REGION Network 49: Step[1021] : Uw Semi Splicer Vacuum Left Bottom HomePos & Right Bottom WorkPos Command
   RUNG wire#powerrail
      { S7_Templates := "SrcType := DInt" } EQ_Contact(in1 := "Unit1.Em2.ControlNodes".SemiAutuSplice.sequence.status.currentStep, in2 := #JOB_10_STEP_21)
      Contact( "Unit1.Em2.ControlNodes".SemiAutuSplice.sequence.status.seqActive )
      wire#w1
      I_Contact( "Unit1.Em2.ControlNodes".cmUwSemiSplicerVacuumRightBottomOnOff.monitoring.inWorkPos )
      Coil( "Unit1.Em2.ControlNodes".SemiAutuSplice."step".action[1021] )
   END_RUNG
   RUNG wire#w1
      Contact( "Unit1.Em2.ControlNodes".cmUwSemiSplicerVacuumRightBottomOnOff.monitoring.inWorkPos )
      wire#w2
      Contact( "Unit1.Em2.ControlNodes".cmUwSemiSplicerVacuumLeftBottomOnOff.monitoring.inWorkPos )
      wire#w3
      Coil( "Unit1.Em2.ControlNodes".SemiAutuSplice."step".action[1022] )
   END_RUNG
   RUNG wire#w1
      Contact( "Unit1.Em2.HmiInterface".cmUwSemiSplicerVacuumRightBottomOnOff.monitoring.goToWorkPos )
   END_RUNG wire#w2
   RUNG wire#w2
      Contact( "Unit1.Em2.HmiInterface".cmUwSemiSplicerVacuumLeftBottomOnOff.monitoring.goToWorkPos )
   END_RUNG wire#w3
   RUNG wire#w1
      Contact( "Unit1.Em2.ControlNodes".cmUwSemiSplicerVacuumRightBottomOnOff.monitoring.inWorkPos )
      Contact( "Unit1.Em2.ControlNodes".cmUwSemiSplicerVacuumLeftBottomOnOff.monitoring.inHomePos )
      Coil( "Unit1.Em2.ControlNodes".SemiAutuSplice."step".transition[1021] )
   END_RUNG
   RUNG wire#w1
      Contact( "Unit1.Em2.ControlNodes".SemiAutuSplice."step".transition[1021] )
      { S7_Templates := "time_type := Time" } #statTonTimer[1021].TON(pt := #SeqDelayTime, et =>)
      Move(in := #STEP_IDLE, out1 => "Unit1.Em2.ControlNodes".SemiAutuSplice.sequence.status.nextStep)
   END_RUNG
   // the same network as SCL:
   #_w1 := ("Unit1.Em2.ControlNodes".SemiAutuSplice.sequence.status.currentStep = #JOB_10_STEP_21) AND "Unit1.Em2.ControlNodes".SemiAutuSplice.sequence.status.seqActive;
   "Unit1.Em2.ControlNodes".SemiAutuSplice."step".action[1021] := #_w1 AND NOT "Unit1.Em2.ControlNodes".cmUwSemiSplicerVacuumRightBottomOnOff.monitoring.inWorkPos;
   "Unit1.Em2.ControlNodes".SemiAutuSplice."step".action[1022] := #_w1 AND ("Unit1.Em2.ControlNodes".cmUwSemiSplicerVacuumRightBottomOnOff.monitoring.inWorkPos OR "Unit1.Em2.HmiInterface".cmUwSemiSplicerVacuumRightBottomOnOff.monitoring.goToWorkPos) AND ("Unit1.Em2.ControlNodes".cmUwSemiSplicerVacuumLeftBottomOnOff.monitoring.inWorkPos OR "Unit1.Em2.HmiInterface".cmUwSemiSplicerVacuumLeftBottomOnOff.monitoring.goToWorkPos);
   "Unit1.Em2.ControlNodes".SemiAutuSplice."step".transition[1021] := #_w1 AND "Unit1.Em2.ControlNodes".cmUwSemiSplicerVacuumRightBottomOnOff.monitoring.inWorkPos AND "Unit1.Em2.ControlNodes".cmUwSemiSplicerVacuumLeftBottomOnOff.monitoring.inHomePos;
   #statTonTimer[1021].TON(IN := #_w1 AND "Unit1.Em2.ControlNodes".SemiAutuSplice."step".transition[1021],
                           PT := #SeqDelayTime);
   IF #statTonTimer[1021].Q THEN
       "Unit1.Em2.ControlNodes".SemiAutuSplice.sequence.status.nextStep := #STEP_IDLE;
   END_IF;
END_REGION

REGION Network 50: ******************** JOB[11] : TAPE ATTACH READY PROCESS AUTO ********************
END_REGION

REGION Network 51: Step[1101] : Electrode Fix Left Top & Electrode Fix Bottom HomePos Command
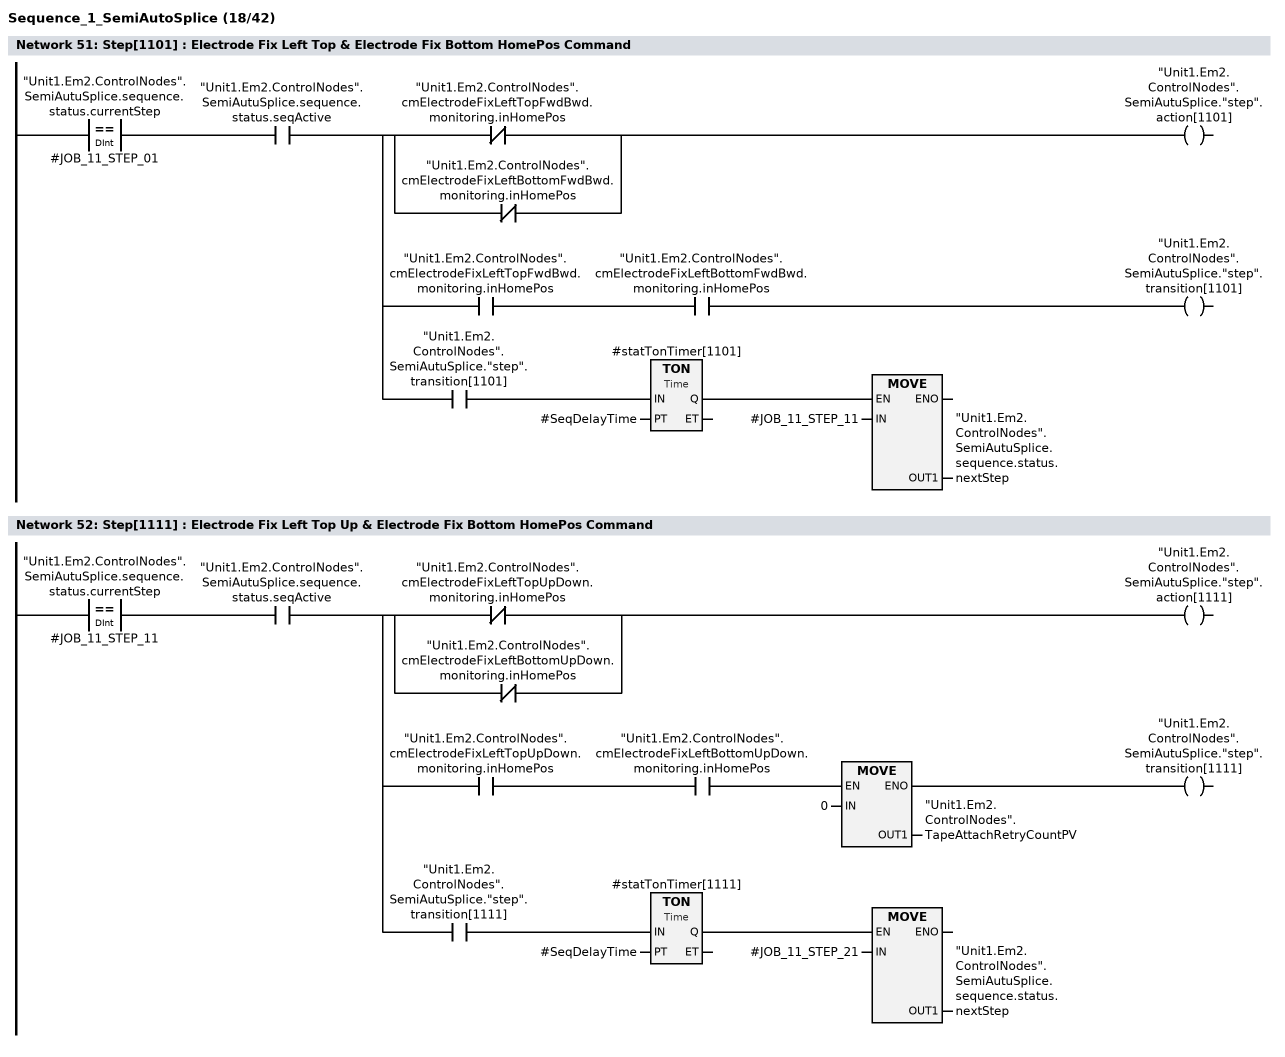
   RUNG wire#powerrail
      { S7_Templates := "SrcType := DInt" } EQ_Contact(in1 := "Unit1.Em2.ControlNodes".SemiAutuSplice.sequence.status.currentStep, in2 := #JOB_11_STEP_01)
      Contact( "Unit1.Em2.ControlNodes".SemiAutuSplice.sequence.status.seqActive )
      wire#w1
      I_Contact( "Unit1.Em2.ControlNodes".cmElectrodeFixLeftTopFwdBwd.monitoring.inHomePos )
      wire#w2
      Coil( "Unit1.Em2.ControlNodes".SemiAutuSplice."step".action[1101] )
   END_RUNG
   RUNG wire#w1
      I_Contact( "Unit1.Em2.ControlNodes".cmElectrodeFixLeftBottomFwdBwd.monitoring.inHomePos )
   END_RUNG wire#w2
   RUNG wire#w1
      Contact( "Unit1.Em2.ControlNodes".cmElectrodeFixLeftTopFwdBwd.monitoring.inHomePos )
      Contact( "Unit1.Em2.ControlNodes".cmElectrodeFixLeftBottomFwdBwd.monitoring.inHomePos )
      Coil( "Unit1.Em2.ControlNodes".SemiAutuSplice."step".transition[1101] )
   END_RUNG
   RUNG wire#w1
      Contact( "Unit1.Em2.ControlNodes".SemiAutuSplice."step".transition[1101] )
      { S7_Templates := "time_type := Time" } #statTonTimer[1101].TON(pt := #SeqDelayTime, et =>)
      Move(in := #JOB_11_STEP_11, out1 => "Unit1.Em2.ControlNodes".SemiAutuSplice.sequence.status.nextStep)
   END_RUNG
   // the same network as SCL:
   #_w1 := ("Unit1.Em2.ControlNodes".SemiAutuSplice.sequence.status.currentStep = #JOB_11_STEP_01) AND "Unit1.Em2.ControlNodes".SemiAutuSplice.sequence.status.seqActive;
   "Unit1.Em2.ControlNodes".SemiAutuSplice."step".action[1101] := #_w1 AND (NOT "Unit1.Em2.ControlNodes".cmElectrodeFixLeftTopFwdBwd.monitoring.inHomePos OR NOT "Unit1.Em2.ControlNodes".cmElectrodeFixLeftBottomFwdBwd.monitoring.inHomePos);
   "Unit1.Em2.ControlNodes".SemiAutuSplice."step".transition[1101] := #_w1 AND "Unit1.Em2.ControlNodes".cmElectrodeFixLeftTopFwdBwd.monitoring.inHomePos AND "Unit1.Em2.ControlNodes".cmElectrodeFixLeftBottomFwdBwd.monitoring.inHomePos;
   #statTonTimer[1101].TON(IN := #_w1 AND "Unit1.Em2.ControlNodes".SemiAutuSplice."step".transition[1101],
                           PT := #SeqDelayTime);
   IF #statTonTimer[1101].Q THEN
       "Unit1.Em2.ControlNodes".SemiAutuSplice.sequence.status.nextStep := #JOB_11_STEP_11;
   END_IF;
END_REGION

REGION Network 52: Step[1111] : Electrode Fix Left Top Up & Electrode Fix Bottom HomePos Command
   RUNG wire#powerrail
      { S7_Templates := "SrcType := DInt" } EQ_Contact(in1 := "Unit1.Em2.ControlNodes".SemiAutuSplice.sequence.status.currentStep, in2 := #JOB_11_STEP_11)
      Contact( "Unit1.Em2.ControlNodes".SemiAutuSplice.sequence.status.seqActive )
      wire#w1
      I_Contact( "Unit1.Em2.ControlNodes".cmElectrodeFixLeftTopUpDown.monitoring.inHomePos )
      wire#w2
      Coil( "Unit1.Em2.ControlNodes".SemiAutuSplice."step".action[1111] )
   END_RUNG
   RUNG wire#w1
      I_Contact( "Unit1.Em2.ControlNodes".cmElectrodeFixLeftBottomUpDown.monitoring.inHomePos )
   END_RUNG wire#w2
   RUNG wire#w1
      Contact( "Unit1.Em2.ControlNodes".cmElectrodeFixLeftTopUpDown.monitoring.inHomePos )
      Contact( "Unit1.Em2.ControlNodes".cmElectrodeFixLeftBottomUpDown.monitoring.inHomePos )
      Move(in := 0, out1 => "Unit1.Em2.ControlNodes".TapeAttachRetryCountPV)
      Coil( "Unit1.Em2.ControlNodes".SemiAutuSplice."step".transition[1111] )
   END_RUNG
   RUNG wire#w1
      Contact( "Unit1.Em2.ControlNodes".SemiAutuSplice."step".transition[1111] )
      { S7_Templates := "time_type := Time" } #statTonTimer[1111].TON(pt := #SeqDelayTime, et =>)
      Move(in := #JOB_11_STEP_21, out1 => "Unit1.Em2.ControlNodes".SemiAutuSplice.sequence.status.nextStep)
   END_RUNG
   // the same network as SCL:
   #_w1 := ("Unit1.Em2.ControlNodes".SemiAutuSplice.sequence.status.currentStep = #JOB_11_STEP_11) AND "Unit1.Em2.ControlNodes".SemiAutuSplice.sequence.status.seqActive;
   "Unit1.Em2.ControlNodes".SemiAutuSplice."step".action[1111] := #_w1 AND (NOT "Unit1.Em2.ControlNodes".cmElectrodeFixLeftTopUpDown.monitoring.inHomePos OR NOT "Unit1.Em2.ControlNodes".cmElectrodeFixLeftBottomUpDown.monitoring.inHomePos);
   #_w2 := #_w1 AND "Unit1.Em2.ControlNodes".cmElectrodeFixLeftTopUpDown.monitoring.inHomePos AND "Unit1.Em2.ControlNodes".cmElectrodeFixLeftBottomUpDown.monitoring.inHomePos;
   IF #_w2 THEN "Unit1.Em2.ControlNodes".TapeAttachRetryCountPV := 0; END_IF;
   "Unit1.Em2.ControlNodes".SemiAutuSplice."step".transition[1111] := #_w2;
   #statTonTimer[1111].TON(IN := #_w1 AND "Unit1.Em2.ControlNodes".SemiAutuSplice."step".transition[1111],
                           PT := #SeqDelayTime);
   IF #statTonTimer[1111].Q THEN
       "Unit1.Em2.ControlNodes".SemiAutuSplice.sequence.status.nextStep := #JOB_11_STEP_21;
   END_IF;
END_REGION

REGION Network 53: Step[1121] : Tape Loading Turn WorkPos Command
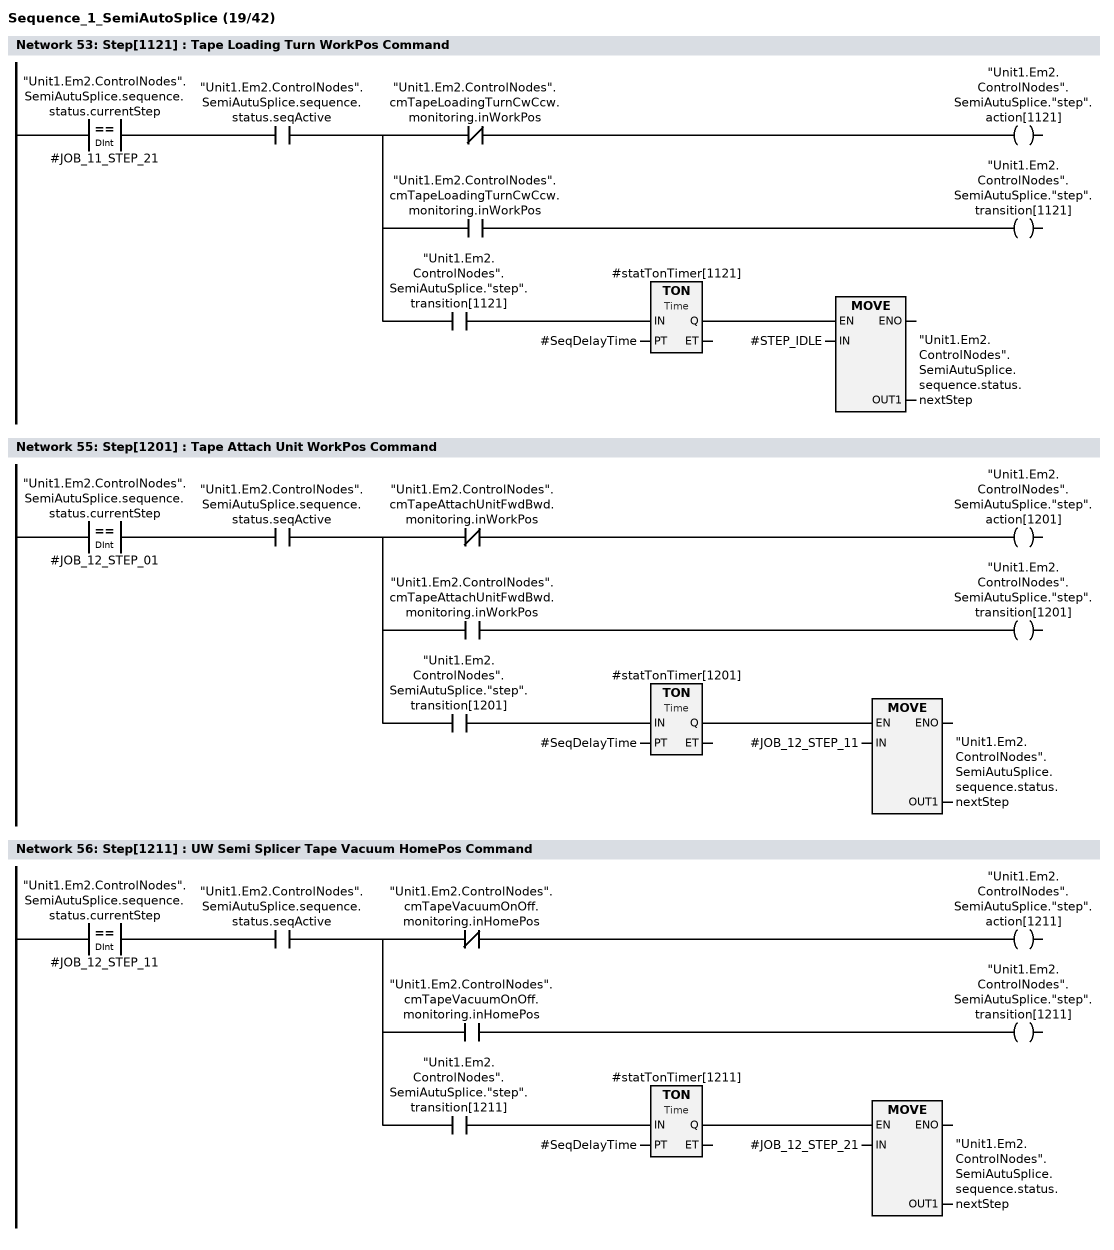
   RUNG wire#powerrail
      { S7_Templates := "SrcType := DInt" } EQ_Contact(in1 := "Unit1.Em2.ControlNodes".SemiAutuSplice.sequence.status.currentStep, in2 := #JOB_11_STEP_21)
      Contact( "Unit1.Em2.ControlNodes".SemiAutuSplice.sequence.status.seqActive )
      wire#w1
      I_Contact( "Unit1.Em2.ControlNodes".cmTapeLoadingTurnCwCcw.monitoring.inWorkPos )
      Coil( "Unit1.Em2.ControlNodes".SemiAutuSplice."step".action[1121] )
   END_RUNG
   RUNG wire#w1
      Contact( "Unit1.Em2.ControlNodes".cmTapeLoadingTurnCwCcw.monitoring.inWorkPos )
      Coil( "Unit1.Em2.ControlNodes".SemiAutuSplice."step".transition[1121] )
   END_RUNG
   RUNG wire#w1
      Contact( "Unit1.Em2.ControlNodes".SemiAutuSplice."step".transition[1121] )
      { S7_Templates := "time_type := Time" } #statTonTimer[1121].TON(pt := #SeqDelayTime, et =>)
      Move(in := #STEP_IDLE, out1 => "Unit1.Em2.ControlNodes".SemiAutuSplice.sequence.status.nextStep)
   END_RUNG
   // the same network as SCL:
   #_w1 := ("Unit1.Em2.ControlNodes".SemiAutuSplice.sequence.status.currentStep = #JOB_11_STEP_21) AND "Unit1.Em2.ControlNodes".SemiAutuSplice.sequence.status.seqActive;
   "Unit1.Em2.ControlNodes".SemiAutuSplice."step".action[1121] := #_w1 AND NOT "Unit1.Em2.ControlNodes".cmTapeLoadingTurnCwCcw.monitoring.inWorkPos;
   "Unit1.Em2.ControlNodes".SemiAutuSplice."step".transition[1121] := #_w1 AND "Unit1.Em2.ControlNodes".cmTapeLoadingTurnCwCcw.monitoring.inWorkPos;
   #statTonTimer[1121].TON(IN := #_w1 AND "Unit1.Em2.ControlNodes".SemiAutuSplice."step".transition[1121],
                           PT := #SeqDelayTime);
   IF #statTonTimer[1121].Q THEN
       "Unit1.Em2.ControlNodes".SemiAutuSplice.sequence.status.nextStep := #STEP_IDLE;
   END_IF;
END_REGION

REGION Network 54: ******************** JOB[12] TAPE ATTACH START PROCESS AUTO ********************
END_REGION

REGION Network 55: Step[1201] : Tape Attach Unit WorkPos Command
   RUNG wire#powerrail
      { S7_Templates := "SrcType := DInt" } EQ_Contact(in1 := "Unit1.Em2.ControlNodes".SemiAutuSplice.sequence.status.currentStep, in2 := #JOB_12_STEP_01)
      Contact( "Unit1.Em2.ControlNodes".SemiAutuSplice.sequence.status.seqActive )
      wire#w1
      I_Contact( "Unit1.Em2.ControlNodes".cmTapeAttachUnitFwdBwd.monitoring.inWorkPos )
      Coil( "Unit1.Em2.ControlNodes".SemiAutuSplice."step".action[1201] )
   END_RUNG
   RUNG wire#w1
      Contact( "Unit1.Em2.ControlNodes".cmTapeAttachUnitFwdBwd.monitoring.inWorkPos )
      Coil( "Unit1.Em2.ControlNodes".SemiAutuSplice."step".transition[1201] )
   END_RUNG
   RUNG wire#w1
      Contact( "Unit1.Em2.ControlNodes".SemiAutuSplice."step".transition[1201] )
      { S7_Templates := "time_type := Time" } #statTonTimer[1201].TON(pt := #SeqDelayTime, et =>)
      Move(in := #JOB_12_STEP_11, out1 => "Unit1.Em2.ControlNodes".SemiAutuSplice.sequence.status.nextStep)
   END_RUNG
   // the same network as SCL:
   #_w1 := ("Unit1.Em2.ControlNodes".SemiAutuSplice.sequence.status.currentStep = #JOB_12_STEP_01) AND "Unit1.Em2.ControlNodes".SemiAutuSplice.sequence.status.seqActive;
   "Unit1.Em2.ControlNodes".SemiAutuSplice."step".action[1201] := #_w1 AND NOT "Unit1.Em2.ControlNodes".cmTapeAttachUnitFwdBwd.monitoring.inWorkPos;
   "Unit1.Em2.ControlNodes".SemiAutuSplice."step".transition[1201] := #_w1 AND "Unit1.Em2.ControlNodes".cmTapeAttachUnitFwdBwd.monitoring.inWorkPos;
   #statTonTimer[1201].TON(IN := #_w1 AND "Unit1.Em2.ControlNodes".SemiAutuSplice."step".transition[1201],
                           PT := #SeqDelayTime);
   IF #statTonTimer[1201].Q THEN
       "Unit1.Em2.ControlNodes".SemiAutuSplice.sequence.status.nextStep := #JOB_12_STEP_11;
   END_IF;
END_REGION

REGION Network 56: Step[1211] : UW Semi Splicer Tape Vacuum HomePos Command
   RUNG wire#powerrail
      { S7_Templates := "SrcType := DInt" } EQ_Contact(in1 := "Unit1.Em2.ControlNodes".SemiAutuSplice.sequence.status.currentStep, in2 := #JOB_12_STEP_11)
      Contact( "Unit1.Em2.ControlNodes".SemiAutuSplice.sequence.status.seqActive )
      wire#w1
      I_Contact( "Unit1.Em2.ControlNodes".cmTapeVacuumOnOff.monitoring.inHomePos )
      Coil( "Unit1.Em2.ControlNodes".SemiAutuSplice."step".action[1211] )
   END_RUNG
   RUNG wire#w1
      Contact( "Unit1.Em2.ControlNodes".cmTapeVacuumOnOff.monitoring.inHomePos )
      Coil( "Unit1.Em2.ControlNodes".SemiAutuSplice."step".transition[1211] )
   END_RUNG
   RUNG wire#w1
      Contact( "Unit1.Em2.ControlNodes".SemiAutuSplice."step".transition[1211] )
      { S7_Templates := "time_type := Time" } #statTonTimer[1211].TON(pt := #SeqDelayTime, et =>)
      Move(in := #JOB_12_STEP_21, out1 => "Unit1.Em2.ControlNodes".SemiAutuSplice.sequence.status.nextStep)
   END_RUNG
   // the same network as SCL:
   #_w1 := ("Unit1.Em2.ControlNodes".SemiAutuSplice.sequence.status.currentStep = #JOB_12_STEP_11) AND "Unit1.Em2.ControlNodes".SemiAutuSplice.sequence.status.seqActive;
   "Unit1.Em2.ControlNodes".SemiAutuSplice."step".action[1211] := #_w1 AND NOT "Unit1.Em2.ControlNodes".cmTapeVacuumOnOff.monitoring.inHomePos;
   "Unit1.Em2.ControlNodes".SemiAutuSplice."step".transition[1211] := #_w1 AND "Unit1.Em2.ControlNodes".cmTapeVacuumOnOff.monitoring.inHomePos;
   #statTonTimer[1211].TON(IN := #_w1 AND "Unit1.Em2.ControlNodes".SemiAutuSplice."step".transition[1211],
                           PT := #SeqDelayTime);
   IF #statTonTimer[1211].Q THEN
       "Unit1.Em2.ControlNodes".SemiAutuSplice.sequence.status.nextStep := #JOB_12_STEP_21;
   END_IF;
END_REGION

REGION Network 57: Step[1221] : Tape Attach Unit HomePos Command
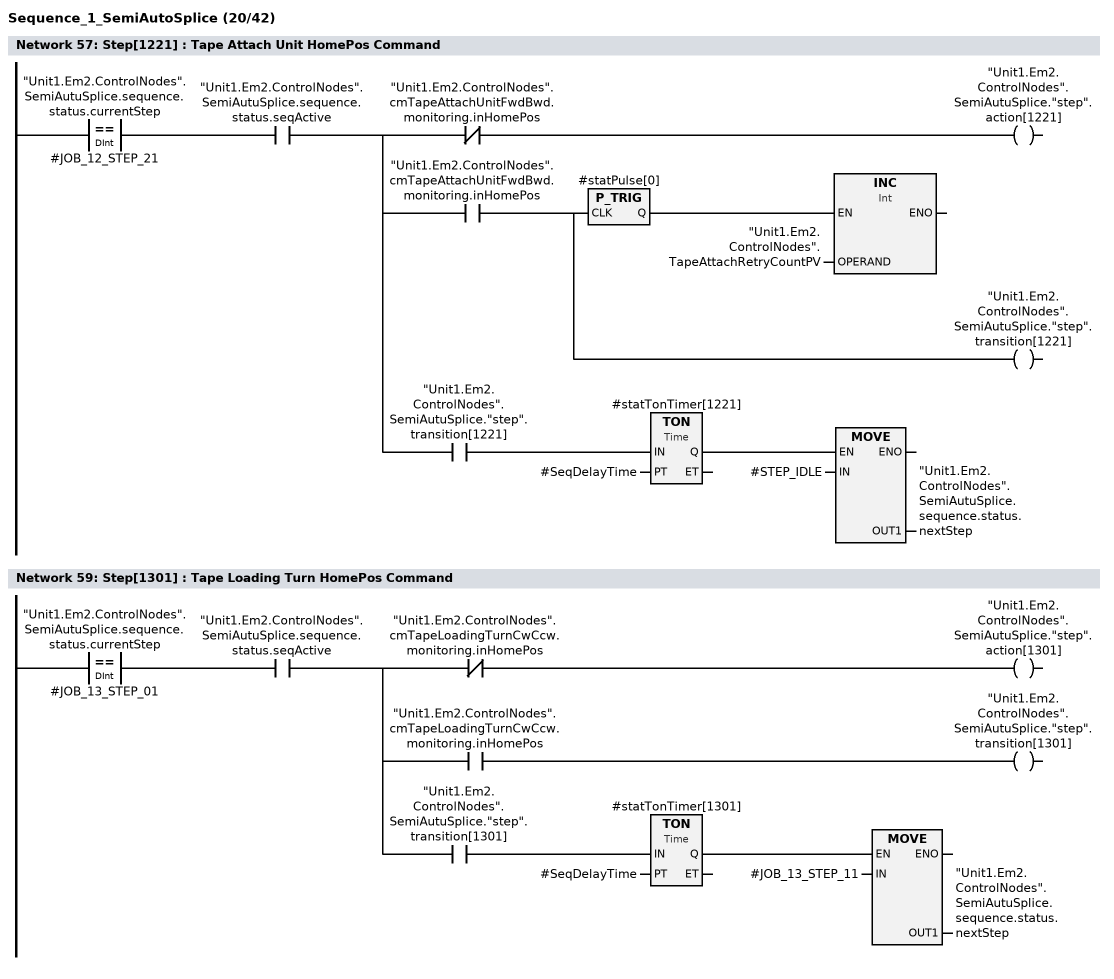
   RUNG wire#powerrail
      { S7_Templates := "SrcType := DInt" } EQ_Contact(in1 := "Unit1.Em2.ControlNodes".SemiAutuSplice.sequence.status.currentStep, in2 := #JOB_12_STEP_21)
      Contact( "Unit1.Em2.ControlNodes".SemiAutuSplice.sequence.status.seqActive )
      wire#w1
      I_Contact( "Unit1.Em2.ControlNodes".cmTapeAttachUnitFwdBwd.monitoring.inHomePos )
      Coil( "Unit1.Em2.ControlNodes".SemiAutuSplice."step".action[1221] )
   END_RUNG
   RUNG wire#w1
      Contact( "Unit1.Em2.ControlNodes".cmTapeAttachUnitFwdBwd.monitoring.inHomePos )
      wire#w2
      P_Trig( #statPulse[0] )
      { S7_Templates := "DestType := Int" } Inc( "Unit1.Em2.ControlNodes".TapeAttachRetryCountPV )
   END_RUNG
   RUNG wire#w2
      Coil( "Unit1.Em2.ControlNodes".SemiAutuSplice."step".transition[1221] )
   END_RUNG
   RUNG wire#w1
      Contact( "Unit1.Em2.ControlNodes".SemiAutuSplice."step".transition[1221] )
      { S7_Templates := "time_type := Time" } #statTonTimer[1221].TON(pt := #SeqDelayTime, et =>)
      Move(in := #STEP_IDLE, out1 => "Unit1.Em2.ControlNodes".SemiAutuSplice.sequence.status.nextStep)
   END_RUNG
   // the same network as SCL:
   #_w1 := ("Unit1.Em2.ControlNodes".SemiAutuSplice.sequence.status.currentStep = #JOB_12_STEP_21) AND "Unit1.Em2.ControlNodes".SemiAutuSplice.sequence.status.seqActive;
   "Unit1.Em2.ControlNodes".SemiAutuSplice."step".action[1221] := #_w1 AND NOT "Unit1.Em2.ControlNodes".cmTapeAttachUnitFwdBwd.monitoring.inHomePos;
   #_w2 := #_w1 AND "Unit1.Em2.ControlNodes".cmTapeAttachUnitFwdBwd.monitoring.inHomePos;
   #_w3 := #_w2 AND NOT #statPulse[0];   // rising edge
   #statPulse[0] := #_w2;
   IF #_w3 THEN
       "Unit1.Em2.ControlNodes".TapeAttachRetryCountPV := "Unit1.Em2.ControlNodes".TapeAttachRetryCountPV + 1;
   END_IF;
   "Unit1.Em2.ControlNodes".SemiAutuSplice."step".transition[1221] := #_w2;
   #statTonTimer[1221].TON(IN := #_w1 AND "Unit1.Em2.ControlNodes".SemiAutuSplice."step".transition[1221],
                           PT := #SeqDelayTime);
   IF #statTonTimer[1221].Q THEN
       "Unit1.Em2.ControlNodes".SemiAutuSplice.sequence.status.nextStep := #STEP_IDLE;
   END_IF;
END_REGION

REGION Network 58: ******************** JOB[13] TAPE ATTACH FINISH PROCESS AUTO ********************
END_REGION

REGION Network 59: Step[1301] : Tape Loading Turn HomePos Command
   RUNG wire#powerrail
      { S7_Templates := "SrcType := DInt" } EQ_Contact(in1 := "Unit1.Em2.ControlNodes".SemiAutuSplice.sequence.status.currentStep, in2 := #JOB_13_STEP_01)
      Contact( "Unit1.Em2.ControlNodes".SemiAutuSplice.sequence.status.seqActive )
      wire#w1
      I_Contact( "Unit1.Em2.ControlNodes".cmTapeLoadingTurnCwCcw.monitoring.inHomePos )
      Coil( "Unit1.Em2.ControlNodes".SemiAutuSplice."step".action[1301] )
   END_RUNG
   RUNG wire#w1
      Contact( "Unit1.Em2.ControlNodes".cmTapeLoadingTurnCwCcw.monitoring.inHomePos )
      Coil( "Unit1.Em2.ControlNodes".SemiAutuSplice."step".transition[1301] )
   END_RUNG
   RUNG wire#w1
      Contact( "Unit1.Em2.ControlNodes".SemiAutuSplice."step".transition[1301] )
      { S7_Templates := "time_type := Time" } #statTonTimer[1301].TON(pt := #SeqDelayTime, et =>)
      Move(in := #JOB_13_STEP_11, out1 => "Unit1.Em2.ControlNodes".SemiAutuSplice.sequence.status.nextStep)
   END_RUNG
   // the same network as SCL:
   #_w1 := ("Unit1.Em2.ControlNodes".SemiAutuSplice.sequence.status.currentStep = #JOB_13_STEP_01) AND "Unit1.Em2.ControlNodes".SemiAutuSplice.sequence.status.seqActive;
   "Unit1.Em2.ControlNodes".SemiAutuSplice."step".action[1301] := #_w1 AND NOT "Unit1.Em2.ControlNodes".cmTapeLoadingTurnCwCcw.monitoring.inHomePos;
   "Unit1.Em2.ControlNodes".SemiAutuSplice."step".transition[1301] := #_w1 AND "Unit1.Em2.ControlNodes".cmTapeLoadingTurnCwCcw.monitoring.inHomePos;
   #statTonTimer[1301].TON(IN := #_w1 AND "Unit1.Em2.ControlNodes".SemiAutuSplice."step".transition[1301],
                           PT := #SeqDelayTime);
   IF #statTonTimer[1301].Q THEN
       "Unit1.Em2.ControlNodes".SemiAutuSplice.sequence.status.nextStep := #JOB_13_STEP_11;
   END_IF;
END_REGION

REGION Network 60: Step[1311] : Uw Semi Splicer Vacuum Right Top & Bottom HomePos Command
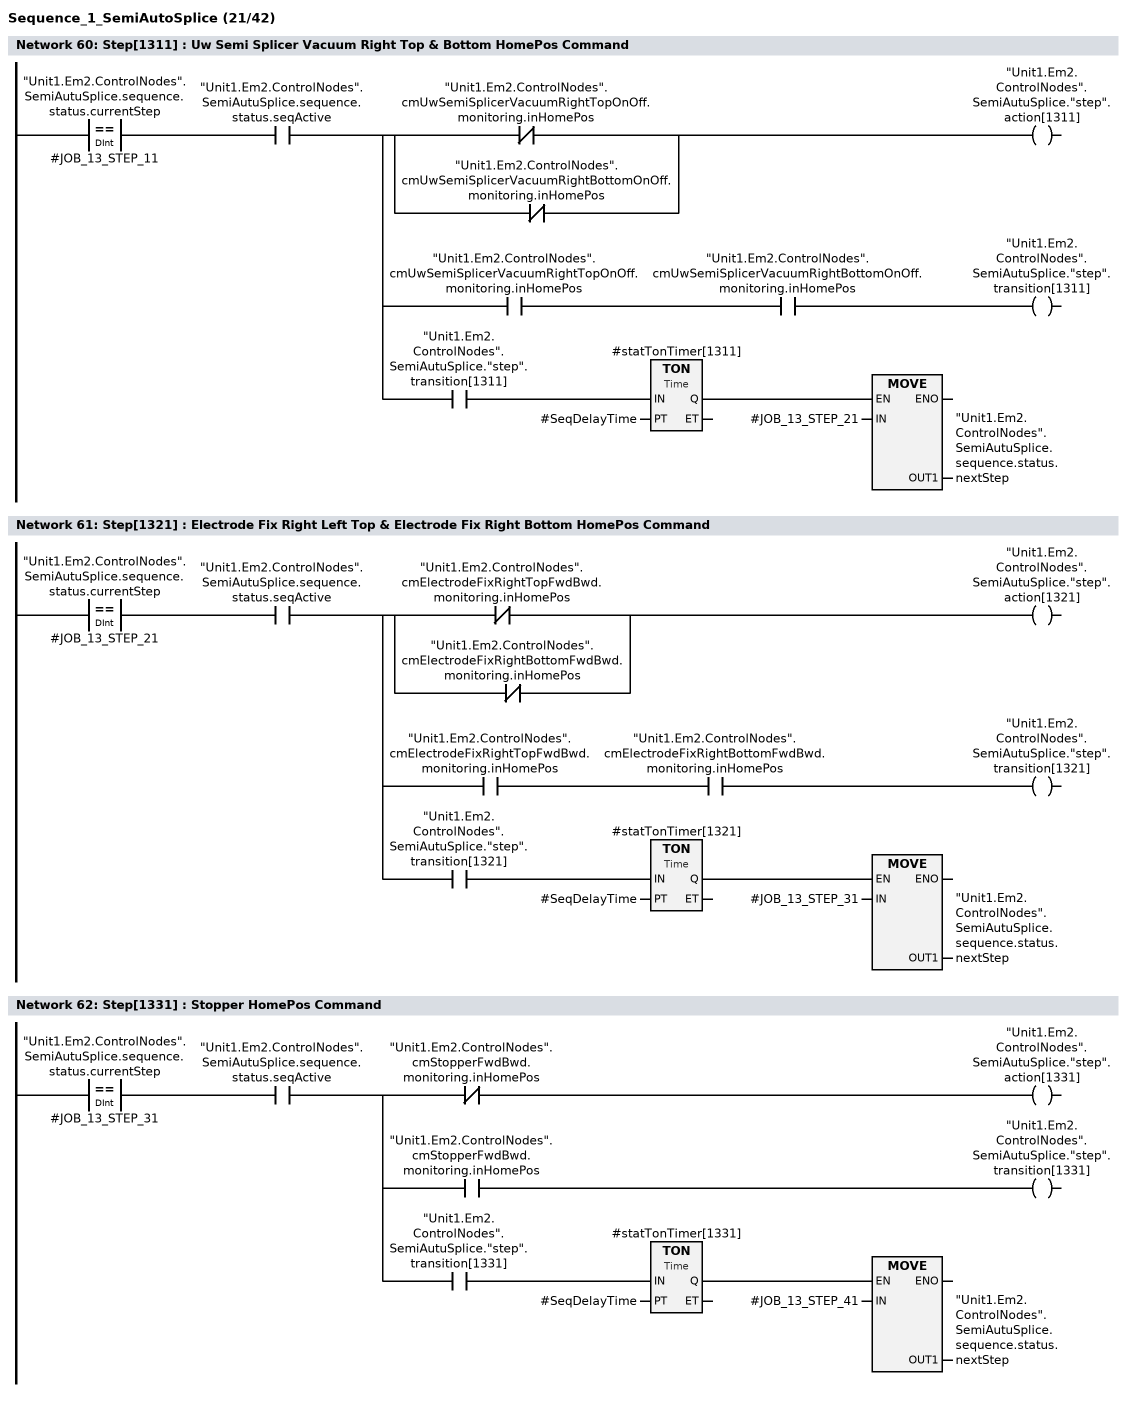
   RUNG wire#powerrail
      { S7_Templates := "SrcType := DInt" } EQ_Contact(in1 := "Unit1.Em2.ControlNodes".SemiAutuSplice.sequence.status.currentStep, in2 := #JOB_13_STEP_11)
      Contact( "Unit1.Em2.ControlNodes".SemiAutuSplice.sequence.status.seqActive )
      wire#w1
      I_Contact( "Unit1.Em2.ControlNodes".cmUwSemiSplicerVacuumRightTopOnOff.monitoring.inHomePos )
      wire#w2
      Coil( "Unit1.Em2.ControlNodes".SemiAutuSplice."step".action[1311] )
   END_RUNG
   RUNG wire#w1
      I_Contact( "Unit1.Em2.ControlNodes".cmUwSemiSplicerVacuumRightBottomOnOff.monitoring.inHomePos )
   END_RUNG wire#w2
   RUNG wire#w1
      Contact( "Unit1.Em2.ControlNodes".cmUwSemiSplicerVacuumRightTopOnOff.monitoring.inHomePos )
      Contact( "Unit1.Em2.ControlNodes".cmUwSemiSplicerVacuumRightBottomOnOff.monitoring.inHomePos )
      Coil( "Unit1.Em2.ControlNodes".SemiAutuSplice."step".transition[1311] )
   END_RUNG
   RUNG wire#w1
      Contact( "Unit1.Em2.ControlNodes".SemiAutuSplice."step".transition[1311] )
      { S7_Templates := "time_type := Time" } #statTonTimer[1311].TON(pt := #SeqDelayTime, et =>)
      Move(in := #JOB_13_STEP_21, out1 => "Unit1.Em2.ControlNodes".SemiAutuSplice.sequence.status.nextStep)
   END_RUNG
   // the same network as SCL:
   #_w1 := ("Unit1.Em2.ControlNodes".SemiAutuSplice.sequence.status.currentStep = #JOB_13_STEP_11) AND "Unit1.Em2.ControlNodes".SemiAutuSplice.sequence.status.seqActive;
   "Unit1.Em2.ControlNodes".SemiAutuSplice."step".action[1311] := #_w1 AND (NOT "Unit1.Em2.ControlNodes".cmUwSemiSplicerVacuumRightTopOnOff.monitoring.inHomePos OR NOT "Unit1.Em2.ControlNodes".cmUwSemiSplicerVacuumRightBottomOnOff.monitoring.inHomePos);
   "Unit1.Em2.ControlNodes".SemiAutuSplice."step".transition[1311] := #_w1 AND "Unit1.Em2.ControlNodes".cmUwSemiSplicerVacuumRightTopOnOff.monitoring.inHomePos AND "Unit1.Em2.ControlNodes".cmUwSemiSplicerVacuumRightBottomOnOff.monitoring.inHomePos;
   #statTonTimer[1311].TON(IN := #_w1 AND "Unit1.Em2.ControlNodes".SemiAutuSplice."step".transition[1311],
                           PT := #SeqDelayTime);
   IF #statTonTimer[1311].Q THEN
       "Unit1.Em2.ControlNodes".SemiAutuSplice.sequence.status.nextStep := #JOB_13_STEP_21;
   END_IF;
END_REGION

REGION Network 61: Step[1321] : Electrode Fix Right Left Top & Electrode Fix Right Bottom HomePos Command
   RUNG wire#powerrail
      { S7_Templates := "SrcType := DInt" } EQ_Contact(in1 := "Unit1.Em2.ControlNodes".SemiAutuSplice.sequence.status.currentStep, in2 := #JOB_13_STEP_21)
      Contact( "Unit1.Em2.ControlNodes".SemiAutuSplice.sequence.status.seqActive )
      wire#w1
      I_Contact( "Unit1.Em2.ControlNodes".cmElectrodeFixRightTopFwdBwd.monitoring.inHomePos )
      wire#w2
      Coil( "Unit1.Em2.ControlNodes".SemiAutuSplice."step".action[1321] )
   END_RUNG
   RUNG wire#w1
      I_Contact( "Unit1.Em2.ControlNodes".cmElectrodeFixRightBottomFwdBwd.monitoring.inHomePos )
   END_RUNG wire#w2
   RUNG wire#w1
      Contact( "Unit1.Em2.ControlNodes".cmElectrodeFixRightTopFwdBwd.monitoring.inHomePos )
      Contact( "Unit1.Em2.ControlNodes".cmElectrodeFixRightBottomFwdBwd.monitoring.inHomePos )
      Coil( "Unit1.Em2.ControlNodes".SemiAutuSplice."step".transition[1321] )
   END_RUNG
   RUNG wire#w1
      Contact( "Unit1.Em2.ControlNodes".SemiAutuSplice."step".transition[1321] )
      { S7_Templates := "time_type := Time" } #statTonTimer[1321].TON(pt := #SeqDelayTime, et =>)
      Move(in := #JOB_13_STEP_31, out1 => "Unit1.Em2.ControlNodes".SemiAutuSplice.sequence.status.nextStep)
   END_RUNG
   // the same network as SCL:
   #_w1 := ("Unit1.Em2.ControlNodes".SemiAutuSplice.sequence.status.currentStep = #JOB_13_STEP_21) AND "Unit1.Em2.ControlNodes".SemiAutuSplice.sequence.status.seqActive;
   "Unit1.Em2.ControlNodes".SemiAutuSplice."step".action[1321] := #_w1 AND (NOT "Unit1.Em2.ControlNodes".cmElectrodeFixRightTopFwdBwd.monitoring.inHomePos OR NOT "Unit1.Em2.ControlNodes".cmElectrodeFixRightBottomFwdBwd.monitoring.inHomePos);
   "Unit1.Em2.ControlNodes".SemiAutuSplice."step".transition[1321] := #_w1 AND "Unit1.Em2.ControlNodes".cmElectrodeFixRightTopFwdBwd.monitoring.inHomePos AND "Unit1.Em2.ControlNodes".cmElectrodeFixRightBottomFwdBwd.monitoring.inHomePos;
   #statTonTimer[1321].TON(IN := #_w1 AND "Unit1.Em2.ControlNodes".SemiAutuSplice."step".transition[1321],
                           PT := #SeqDelayTime);
   IF #statTonTimer[1321].Q THEN
       "Unit1.Em2.ControlNodes".SemiAutuSplice.sequence.status.nextStep := #JOB_13_STEP_31;
   END_IF;
END_REGION

REGION Network 62: Step[1331] : Stopper HomePos Command
   RUNG wire#powerrail
      { S7_Templates := "SrcType := DInt" } EQ_Contact(in1 := "Unit1.Em2.ControlNodes".SemiAutuSplice.sequence.status.currentStep, in2 := #JOB_13_STEP_31)
      Contact( "Unit1.Em2.ControlNodes".SemiAutuSplice.sequence.status.seqActive )
      wire#w1
      I_Contact( "Unit1.Em2.ControlNodes".cmStopperFwdBwd.monitoring.inHomePos )
      Coil( "Unit1.Em2.ControlNodes".SemiAutuSplice."step".action[1331] )
   END_RUNG
   RUNG wire#w1
      Contact( "Unit1.Em2.ControlNodes".cmStopperFwdBwd.monitoring.inHomePos )
      Coil( "Unit1.Em2.ControlNodes".SemiAutuSplice."step".transition[1331] )
   END_RUNG
   RUNG wire#w1
      Contact( "Unit1.Em2.ControlNodes".SemiAutuSplice."step".transition[1331] )
      { S7_Templates := "time_type := Time" } #statTonTimer[1331].TON(pt := #SeqDelayTime, et =>)
      Move(in := #JOB_13_STEP_41, out1 => "Unit1.Em2.ControlNodes".SemiAutuSplice.sequence.status.nextStep)
   END_RUNG
   // the same network as SCL:
   #_w1 := ("Unit1.Em2.ControlNodes".SemiAutuSplice.sequence.status.currentStep = #JOB_13_STEP_31) AND "Unit1.Em2.ControlNodes".SemiAutuSplice.sequence.status.seqActive;
   "Unit1.Em2.ControlNodes".SemiAutuSplice."step".action[1331] := #_w1 AND NOT "Unit1.Em2.ControlNodes".cmStopperFwdBwd.monitoring.inHomePos;
   "Unit1.Em2.ControlNodes".SemiAutuSplice."step".transition[1331] := #_w1 AND "Unit1.Em2.ControlNodes".cmStopperFwdBwd.monitoring.inHomePos;
   #statTonTimer[1331].TON(IN := #_w1 AND "Unit1.Em2.ControlNodes".SemiAutuSplice."step".transition[1331],
                           PT := #SeqDelayTime);
   IF #statTonTimer[1331].Q THEN
       "Unit1.Em2.ControlNodes".SemiAutuSplice.sequence.status.nextStep := #JOB_13_STEP_41;
   END_IF;
END_REGION

REGION Network 63: Step[1341] : EM Link Change Check
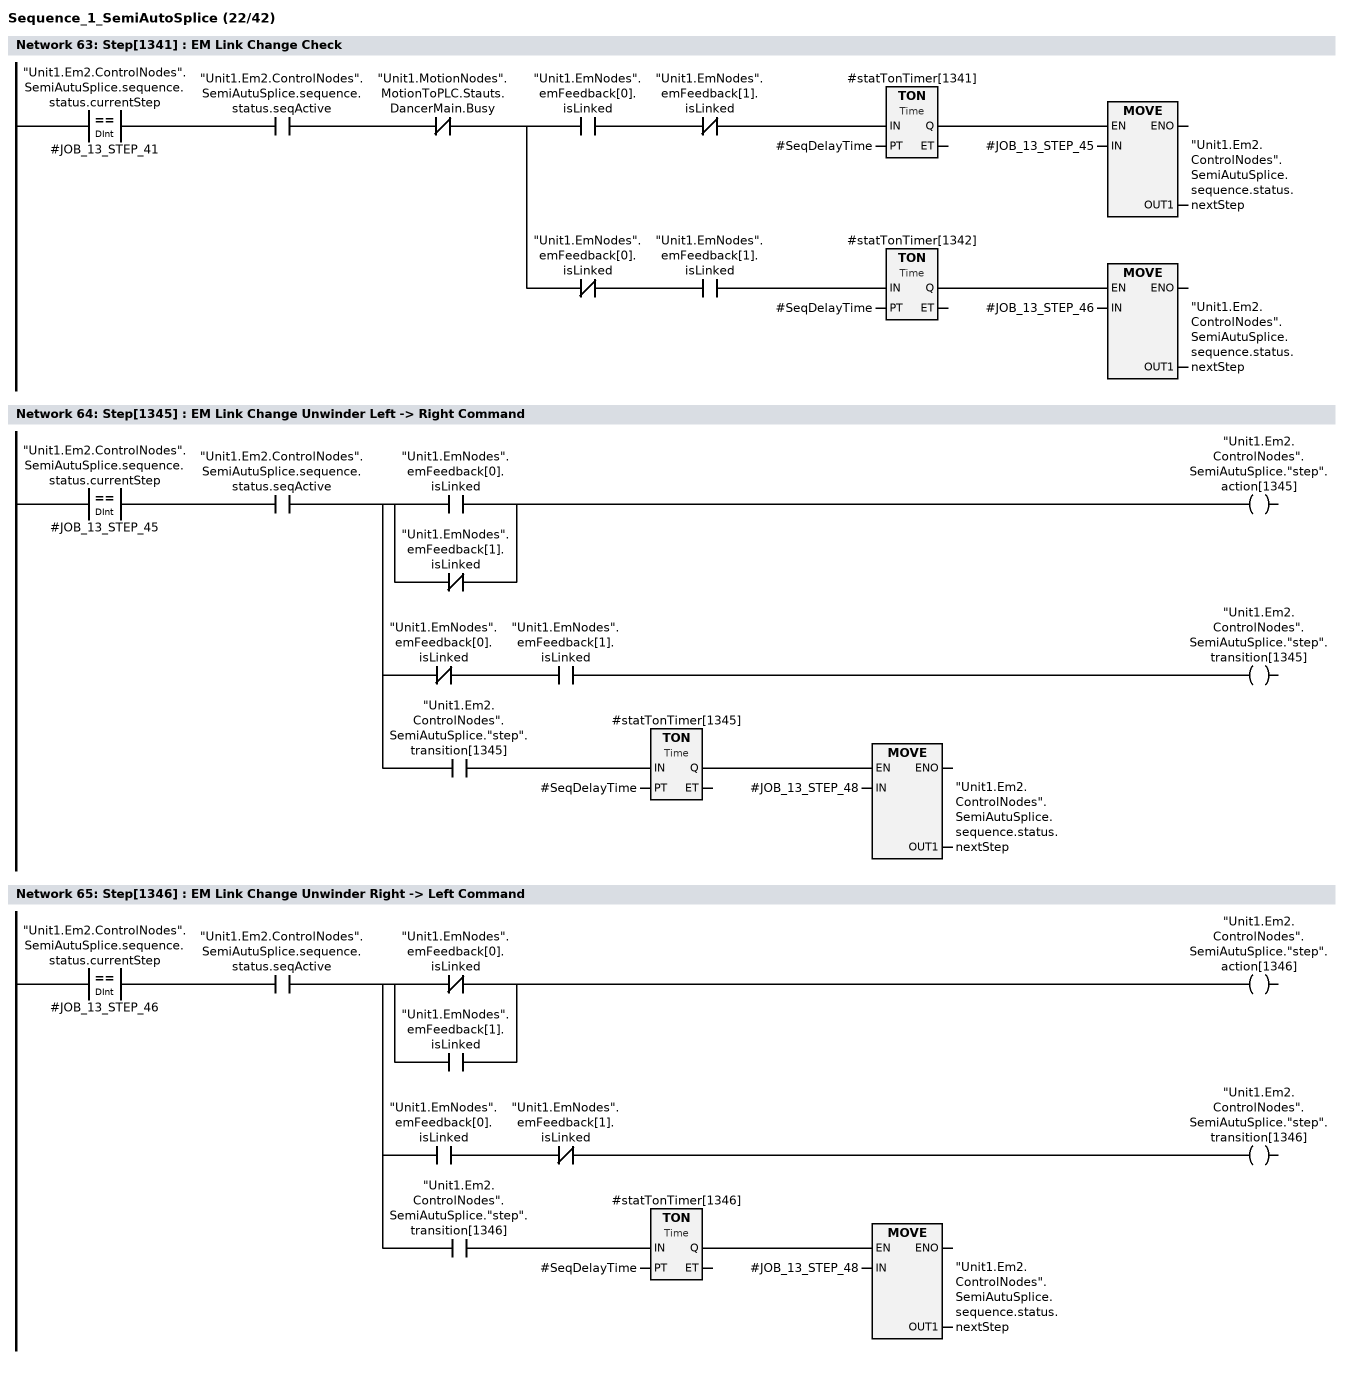
   RUNG wire#powerrail
      { S7_Templates := "SrcType := DInt" } EQ_Contact(in1 := "Unit1.Em2.ControlNodes".SemiAutuSplice.sequence.status.currentStep, in2 := #JOB_13_STEP_41)
      Contact( "Unit1.Em2.ControlNodes".SemiAutuSplice.sequence.status.seqActive )
      I_Contact( "Unit1.MotionNodes".MotionToPLC.Stauts.DancerMain.Busy )
      wire#w1
      Contact( "Unit1.EmNodes".emFeedback[0].isLinked )
      I_Contact( "Unit1.EmNodes".emFeedback[1].isLinked )
      { S7_Templates := "time_type := Time" } #statTonTimer[1341].TON(pt := #SeqDelayTime, et =>)
      Move(in := #JOB_13_STEP_45, out1 => "Unit1.Em2.ControlNodes".SemiAutuSplice.sequence.status.nextStep)
   END_RUNG
   RUNG wire#w1
      I_Contact( "Unit1.EmNodes".emFeedback[0].isLinked )
      Contact( "Unit1.EmNodes".emFeedback[1].isLinked )
      { S7_Templates := "time_type := Time" } #statTonTimer[1342].TON(pt := #SeqDelayTime, et =>)
      Move(in := #JOB_13_STEP_46, out1 => "Unit1.Em2.ControlNodes".SemiAutuSplice.sequence.status.nextStep)
   END_RUNG
   // the same network as SCL:
   #_w1 := ("Unit1.Em2.ControlNodes".SemiAutuSplice.sequence.status.currentStep = #JOB_13_STEP_41) AND "Unit1.Em2.ControlNodes".SemiAutuSplice.sequence.status.seqActive AND NOT "Unit1.MotionNodes".MotionToPLC.Stauts.DancerMain.Busy;
   #statTonTimer[1341].TON(IN := #_w1 AND "Unit1.EmNodes".emFeedback[0].isLinked AND NOT "Unit1.EmNodes".emFeedback[1].isLinked,
                           PT := #SeqDelayTime);
   IF #statTonTimer[1341].Q THEN
       "Unit1.Em2.ControlNodes".SemiAutuSplice.sequence.status.nextStep := #JOB_13_STEP_45;
   END_IF;
   #statTonTimer[1342].TON(IN := #_w1 AND NOT "Unit1.EmNodes".emFeedback[0].isLinked AND "Unit1.EmNodes".emFeedback[1].isLinked,
                           PT := #SeqDelayTime);
   IF #statTonTimer[1342].Q THEN
       "Unit1.Em2.ControlNodes".SemiAutuSplice.sequence.status.nextStep := #JOB_13_STEP_46;
   END_IF;
END_REGION

REGION Network 64: Step[1345] : EM Link Change Unwinder Left -> Right Command
   RUNG wire#powerrail
      { S7_Templates := "SrcType := DInt" } EQ_Contact(in1 := "Unit1.Em2.ControlNodes".SemiAutuSplice.sequence.status.currentStep, in2 := #JOB_13_STEP_45)
      Contact( "Unit1.Em2.ControlNodes".SemiAutuSplice.sequence.status.seqActive )
      wire#w1
      Contact( "Unit1.EmNodes".emFeedback[0].isLinked )
      wire#w2
      Coil( "Unit1.Em2.ControlNodes".SemiAutuSplice."step".action[1345] )
   END_RUNG
   RUNG wire#w1
      I_Contact( "Unit1.EmNodes".emFeedback[1].isLinked )
   END_RUNG wire#w2
   RUNG wire#w1
      I_Contact( "Unit1.EmNodes".emFeedback[0].isLinked )
      Contact( "Unit1.EmNodes".emFeedback[1].isLinked )
      Coil( "Unit1.Em2.ControlNodes".SemiAutuSplice."step".transition[1345] )
   END_RUNG
   RUNG wire#w1
      Contact( "Unit1.Em2.ControlNodes".SemiAutuSplice."step".transition[1345] )
      { S7_Templates := "time_type := Time" } #statTonTimer[1345].TON(pt := #SeqDelayTime, et =>)
      Move(in := #JOB_13_STEP_48, out1 => "Unit1.Em2.ControlNodes".SemiAutuSplice.sequence.status.nextStep)
   END_RUNG
   // the same network as SCL:
   #_w1 := ("Unit1.Em2.ControlNodes".SemiAutuSplice.sequence.status.currentStep = #JOB_13_STEP_45) AND "Unit1.Em2.ControlNodes".SemiAutuSplice.sequence.status.seqActive;
   "Unit1.Em2.ControlNodes".SemiAutuSplice."step".action[1345] := #_w1 AND ("Unit1.EmNodes".emFeedback[0].isLinked OR NOT "Unit1.EmNodes".emFeedback[1].isLinked);
   "Unit1.Em2.ControlNodes".SemiAutuSplice."step".transition[1345] := #_w1 AND NOT "Unit1.EmNodes".emFeedback[0].isLinked AND "Unit1.EmNodes".emFeedback[1].isLinked;
   #statTonTimer[1345].TON(IN := #_w1 AND "Unit1.Em2.ControlNodes".SemiAutuSplice."step".transition[1345],
                           PT := #SeqDelayTime);
   IF #statTonTimer[1345].Q THEN
       "Unit1.Em2.ControlNodes".SemiAutuSplice.sequence.status.nextStep := #JOB_13_STEP_48;
   END_IF;
END_REGION

REGION Network 65: Step[1346] : EM Link Change Unwinder Right -> Left Command
   RUNG wire#powerrail
      { S7_Templates := "SrcType := DInt" } EQ_Contact(in1 := "Unit1.Em2.ControlNodes".SemiAutuSplice.sequence.status.currentStep, in2 := #JOB_13_STEP_46)
      Contact( "Unit1.Em2.ControlNodes".SemiAutuSplice.sequence.status.seqActive )
      wire#w1
      I_Contact( "Unit1.EmNodes".emFeedback[0].isLinked )
      wire#w2
      Coil( "Unit1.Em2.ControlNodes".SemiAutuSplice."step".action[1346] )
   END_RUNG
   RUNG wire#w1
      Contact( "Unit1.EmNodes".emFeedback[1].isLinked )
   END_RUNG wire#w2
   RUNG wire#w1
      Contact( "Unit1.EmNodes".emFeedback[0].isLinked )
      I_Contact( "Unit1.EmNodes".emFeedback[1].isLinked )
      Coil( "Unit1.Em2.ControlNodes".SemiAutuSplice."step".transition[1346] )
   END_RUNG
   RUNG wire#w1
      Contact( "Unit1.Em2.ControlNodes".SemiAutuSplice."step".transition[1346] )
      { S7_Templates := "time_type := Time" } #statTonTimer[1346].TON(pt := #SeqDelayTime, et =>)
      Move(in := #JOB_13_STEP_48, out1 => "Unit1.Em2.ControlNodes".SemiAutuSplice.sequence.status.nextStep)
   END_RUNG
   // the same network as SCL:
   #_w1 := ("Unit1.Em2.ControlNodes".SemiAutuSplice.sequence.status.currentStep = #JOB_13_STEP_46) AND "Unit1.Em2.ControlNodes".SemiAutuSplice.sequence.status.seqActive;
   "Unit1.Em2.ControlNodes".SemiAutuSplice."step".action[1346] := #_w1 AND (NOT "Unit1.EmNodes".emFeedback[0].isLinked OR "Unit1.EmNodes".emFeedback[1].isLinked);
   "Unit1.Em2.ControlNodes".SemiAutuSplice."step".transition[1346] := #_w1 AND "Unit1.EmNodes".emFeedback[0].isLinked AND NOT "Unit1.EmNodes".emFeedback[1].isLinked;
   #statTonTimer[1346].TON(IN := #_w1 AND "Unit1.Em2.ControlNodes".SemiAutuSplice."step".transition[1346],
                           PT := #SeqDelayTime);
   IF #statTonTimer[1346].Q THEN
       "Unit1.Em2.ControlNodes".SemiAutuSplice.sequence.status.nextStep := #JOB_13_STEP_48;
   END_IF;
END_REGION

REGION Network 66: Step[1348] : EM Link Change Comp
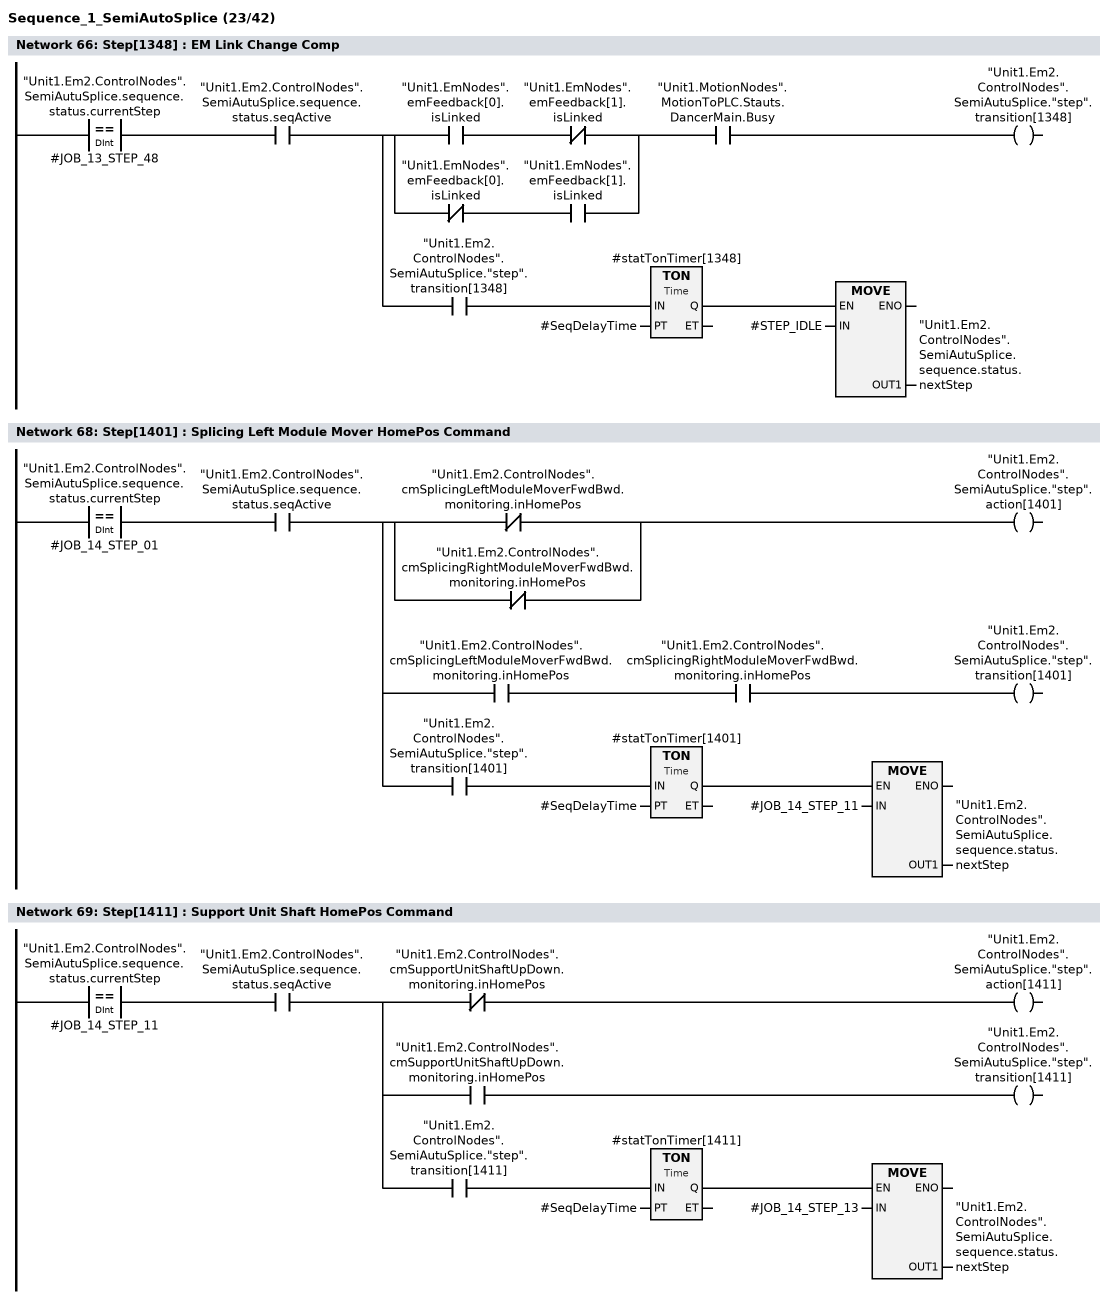
   RUNG wire#powerrail
      { S7_Templates := "SrcType := DInt" } EQ_Contact(in1 := "Unit1.Em2.ControlNodes".SemiAutuSplice.sequence.status.currentStep, in2 := #JOB_13_STEP_48)
      Contact( "Unit1.Em2.ControlNodes".SemiAutuSplice.sequence.status.seqActive )
      wire#w1
      Contact( "Unit1.EmNodes".emFeedback[0].isLinked )
      I_Contact( "Unit1.EmNodes".emFeedback[1].isLinked )
      wire#w2
      Contact( "Unit1.MotionNodes".MotionToPLC.Stauts.DancerMain.Busy )
      Coil( "Unit1.Em2.ControlNodes".SemiAutuSplice."step".transition[1348] )
   END_RUNG
   RUNG wire#w1
      I_Contact( "Unit1.EmNodes".emFeedback[0].isLinked )
      Contact( "Unit1.EmNodes".emFeedback[1].isLinked )
   END_RUNG wire#w2
   RUNG wire#w1
      Contact( "Unit1.Em2.ControlNodes".SemiAutuSplice."step".transition[1348] )
      { S7_Templates := "time_type := Time" } #statTonTimer[1348].TON(pt := #SeqDelayTime, et =>)
      Move(in := #STEP_IDLE, out1 => "Unit1.Em2.ControlNodes".SemiAutuSplice.sequence.status.nextStep)
   END_RUNG
   // the same network as SCL:
   #_w1 := ("Unit1.Em2.ControlNodes".SemiAutuSplice.sequence.status.currentStep = #JOB_13_STEP_48) AND "Unit1.Em2.ControlNodes".SemiAutuSplice.sequence.status.seqActive;
   "Unit1.Em2.ControlNodes".SemiAutuSplice."step".transition[1348] := #_w1 AND (("Unit1.EmNodes".emFeedback[0].isLinked AND NOT "Unit1.EmNodes".emFeedback[1].isLinked) OR (NOT "Unit1.EmNodes".emFeedback[0].isLinked AND "Unit1.EmNodes".emFeedback[1].isLinked)) AND "Unit1.MotionNodes".MotionToPLC.Stauts.DancerMain.Busy;
   #statTonTimer[1348].TON(IN := #_w1 AND "Unit1.Em2.ControlNodes".SemiAutuSplice."step".transition[1348],
                           PT := #SeqDelayTime);
   IF #statTonTimer[1348].Q THEN
       "Unit1.Em2.ControlNodes".SemiAutuSplice.sequence.status.nextStep := #STEP_IDLE;
   END_IF;
END_REGION

REGION Network 67: ******************** JOB[14] LEFT SPLICING MODULE MOVER AUTO ********************
END_REGION

REGION Network 68: Step[1401] : Splicing Left Module Mover HomePos Command
   RUNG wire#powerrail
      { S7_Templates := "SrcType := DInt" } EQ_Contact(in1 := "Unit1.Em2.ControlNodes".SemiAutuSplice.sequence.status.currentStep, in2 := #JOB_14_STEP_01)
      Contact( "Unit1.Em2.ControlNodes".SemiAutuSplice.sequence.status.seqActive )
      wire#w1
      I_Contact( "Unit1.Em2.ControlNodes".cmSplicingLeftModuleMoverFwdBwd.monitoring.inHomePos )
      wire#w2
      Coil( "Unit1.Em2.ControlNodes".SemiAutuSplice."step".action[1401] )
   END_RUNG
   RUNG wire#w1
      I_Contact( "Unit1.Em2.ControlNodes".cmSplicingRightModuleMoverFwdBwd.monitoring.inHomePos )
   END_RUNG wire#w2
   RUNG wire#w1
      Contact( "Unit1.Em2.ControlNodes".cmSplicingLeftModuleMoverFwdBwd.monitoring.inHomePos )
      Contact( "Unit1.Em2.ControlNodes".cmSplicingRightModuleMoverFwdBwd.monitoring.inHomePos )
      Coil( "Unit1.Em2.ControlNodes".SemiAutuSplice."step".transition[1401] )
   END_RUNG
   RUNG wire#w1
      Contact( "Unit1.Em2.ControlNodes".SemiAutuSplice."step".transition[1401] )
      { S7_Templates := "time_type := Time" } #statTonTimer[1401].TON(pt := #SeqDelayTime, et =>)
      Move(in := #JOB_14_STEP_11, out1 => "Unit1.Em2.ControlNodes".SemiAutuSplice.sequence.status.nextStep)
   END_RUNG
   // the same network as SCL:
   #_w1 := ("Unit1.Em2.ControlNodes".SemiAutuSplice.sequence.status.currentStep = #JOB_14_STEP_01) AND "Unit1.Em2.ControlNodes".SemiAutuSplice.sequence.status.seqActive;
   "Unit1.Em2.ControlNodes".SemiAutuSplice."step".action[1401] := #_w1 AND (NOT "Unit1.Em2.ControlNodes".cmSplicingLeftModuleMoverFwdBwd.monitoring.inHomePos OR NOT "Unit1.Em2.ControlNodes".cmSplicingRightModuleMoverFwdBwd.monitoring.inHomePos);
   "Unit1.Em2.ControlNodes".SemiAutuSplice."step".transition[1401] := #_w1 AND "Unit1.Em2.ControlNodes".cmSplicingLeftModuleMoverFwdBwd.monitoring.inHomePos AND "Unit1.Em2.ControlNodes".cmSplicingRightModuleMoverFwdBwd.monitoring.inHomePos;
   #statTonTimer[1401].TON(IN := #_w1 AND "Unit1.Em2.ControlNodes".SemiAutuSplice."step".transition[1401],
                           PT := #SeqDelayTime);
   IF #statTonTimer[1401].Q THEN
       "Unit1.Em2.ControlNodes".SemiAutuSplice.sequence.status.nextStep := #JOB_14_STEP_11;
   END_IF;
END_REGION

REGION Network 69: Step[1411] : Support Unit Shaft HomePos Command
   RUNG wire#powerrail
      { S7_Templates := "SrcType := DInt" } EQ_Contact(in1 := "Unit1.Em2.ControlNodes".SemiAutuSplice.sequence.status.currentStep, in2 := #JOB_14_STEP_11)
      Contact( "Unit1.Em2.ControlNodes".SemiAutuSplice.sequence.status.seqActive )
      wire#w1
      I_Contact( "Unit1.Em2.ControlNodes".cmSupportUnitShaftUpDown.monitoring.inHomePos )
      Coil( "Unit1.Em2.ControlNodes".SemiAutuSplice."step".action[1411] )
   END_RUNG
   RUNG wire#w1
      Contact( "Unit1.Em2.ControlNodes".cmSupportUnitShaftUpDown.monitoring.inHomePos )
      Coil( "Unit1.Em2.ControlNodes".SemiAutuSplice."step".transition[1411] )
   END_RUNG
   RUNG wire#w1
      Contact( "Unit1.Em2.ControlNodes".SemiAutuSplice."step".transition[1411] )
      { S7_Templates := "time_type := Time" } #statTonTimer[1411].TON(pt := #SeqDelayTime, et =>)
      Move(in := #JOB_14_STEP_13, out1 => "Unit1.Em2.ControlNodes".SemiAutuSplice.sequence.status.nextStep)
   END_RUNG
   // the same network as SCL:
   #_w1 := ("Unit1.Em2.ControlNodes".SemiAutuSplice.sequence.status.currentStep = #JOB_14_STEP_11) AND "Unit1.Em2.ControlNodes".SemiAutuSplice.sequence.status.seqActive;
   "Unit1.Em2.ControlNodes".SemiAutuSplice."step".action[1411] := #_w1 AND NOT "Unit1.Em2.ControlNodes".cmSupportUnitShaftUpDown.monitoring.inHomePos;
   "Unit1.Em2.ControlNodes".SemiAutuSplice."step".transition[1411] := #_w1 AND "Unit1.Em2.ControlNodes".cmSupportUnitShaftUpDown.monitoring.inHomePos;
   #statTonTimer[1411].TON(IN := #_w1 AND "Unit1.Em2.ControlNodes".SemiAutuSplice."step".transition[1411],
                           PT := #SeqDelayTime);
   IF #statTonTimer[1411].Q THEN
       "Unit1.Em2.ControlNodes".SemiAutuSplice.sequence.status.nextStep := #JOB_14_STEP_13;
   END_IF;
END_REGION

REGION Network 70: Step[1413] : FrameCover HomePos Command
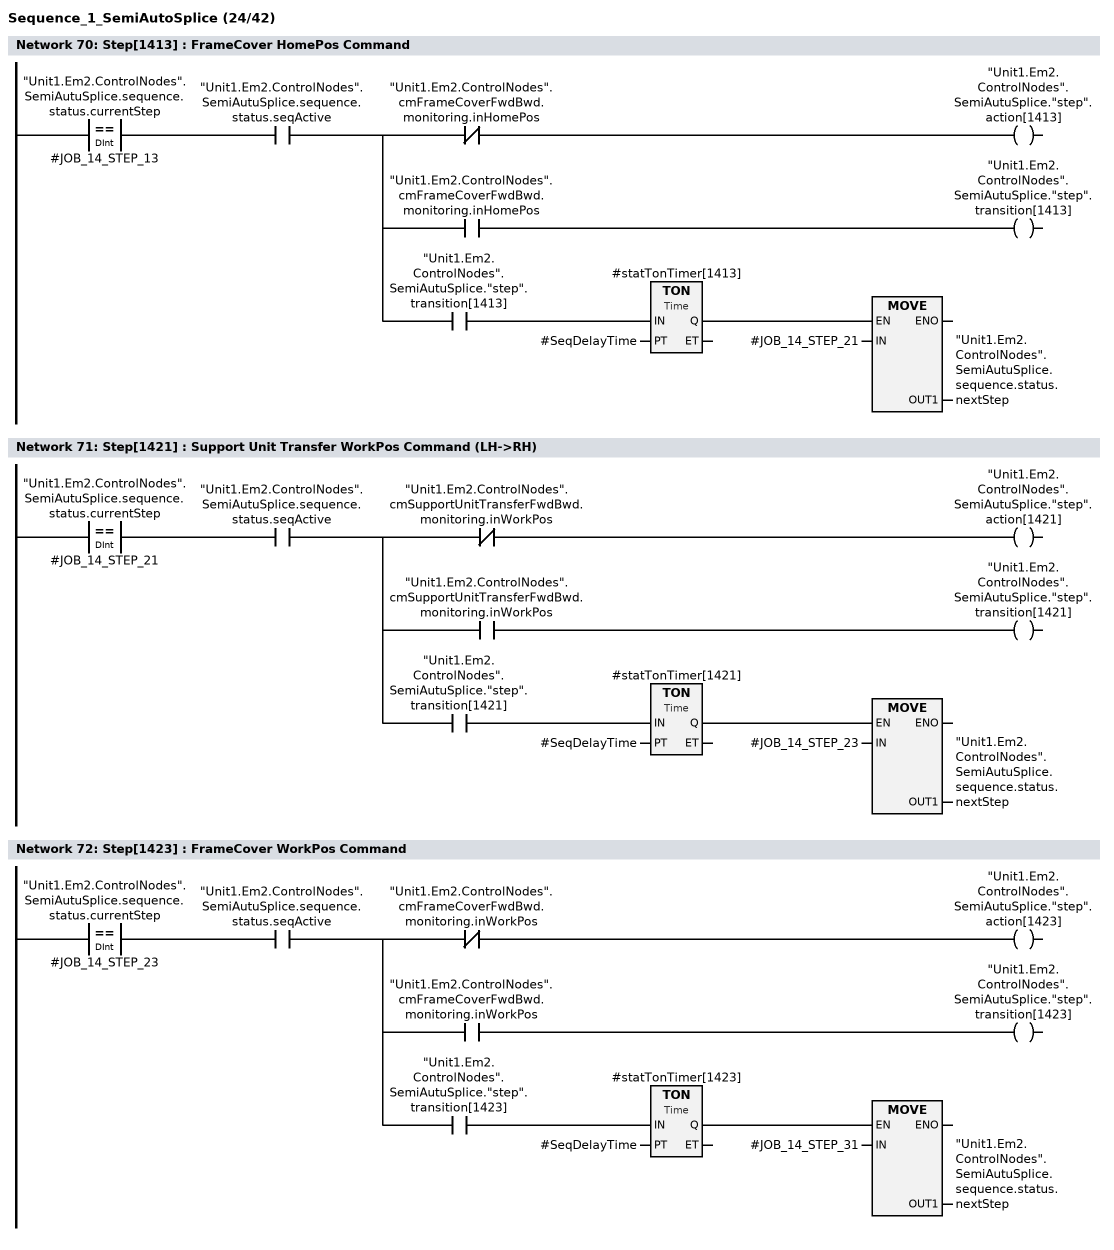
   RUNG wire#powerrail
      { S7_Templates := "SrcType := DInt" } EQ_Contact(in1 := "Unit1.Em2.ControlNodes".SemiAutuSplice.sequence.status.currentStep, in2 := #JOB_14_STEP_13)
      Contact( "Unit1.Em2.ControlNodes".SemiAutuSplice.sequence.status.seqActive )
      wire#w1
      I_Contact( "Unit1.Em2.ControlNodes".cmFrameCoverFwdBwd.monitoring.inHomePos )
      Coil( "Unit1.Em2.ControlNodes".SemiAutuSplice."step".action[1413] )
   END_RUNG
   RUNG wire#w1
      Contact( "Unit1.Em2.ControlNodes".cmFrameCoverFwdBwd.monitoring.inHomePos )
      Coil( "Unit1.Em2.ControlNodes".SemiAutuSplice."step".transition[1413] )
   END_RUNG
   RUNG wire#w1
      Contact( "Unit1.Em2.ControlNodes".SemiAutuSplice."step".transition[1413] )
      { S7_Templates := "time_type := Time" } #statTonTimer[1413].TON(pt := #SeqDelayTime, et =>)
      Move(in := #JOB_14_STEP_21, out1 => "Unit1.Em2.ControlNodes".SemiAutuSplice.sequence.status.nextStep)
   END_RUNG
   // the same network as SCL:
   #_w1 := ("Unit1.Em2.ControlNodes".SemiAutuSplice.sequence.status.currentStep = #JOB_14_STEP_13) AND "Unit1.Em2.ControlNodes".SemiAutuSplice.sequence.status.seqActive;
   "Unit1.Em2.ControlNodes".SemiAutuSplice."step".action[1413] := #_w1 AND NOT "Unit1.Em2.ControlNodes".cmFrameCoverFwdBwd.monitoring.inHomePos;
   "Unit1.Em2.ControlNodes".SemiAutuSplice."step".transition[1413] := #_w1 AND "Unit1.Em2.ControlNodes".cmFrameCoverFwdBwd.monitoring.inHomePos;
   #statTonTimer[1413].TON(IN := #_w1 AND "Unit1.Em2.ControlNodes".SemiAutuSplice."step".transition[1413],
                           PT := #SeqDelayTime);
   IF #statTonTimer[1413].Q THEN
       "Unit1.Em2.ControlNodes".SemiAutuSplice.sequence.status.nextStep := #JOB_14_STEP_21;
   END_IF;
END_REGION

REGION Network 71: Step[1421] : Support Unit Transfer WorkPos Command (LH->RH)
   RUNG wire#powerrail
      { S7_Templates := "SrcType := DInt" } EQ_Contact(in1 := "Unit1.Em2.ControlNodes".SemiAutuSplice.sequence.status.currentStep, in2 := #JOB_14_STEP_21)
      Contact( "Unit1.Em2.ControlNodes".SemiAutuSplice.sequence.status.seqActive )
      wire#w1
      I_Contact( "Unit1.Em2.ControlNodes".cmSupportUnitTransferFwdBwd.monitoring.inWorkPos )
      Coil( "Unit1.Em2.ControlNodes".SemiAutuSplice."step".action[1421] )
   END_RUNG
   RUNG wire#w1
      Contact( "Unit1.Em2.ControlNodes".cmSupportUnitTransferFwdBwd.monitoring.inWorkPos )
      Coil( "Unit1.Em2.ControlNodes".SemiAutuSplice."step".transition[1421] )
   END_RUNG
   RUNG wire#w1
      Contact( "Unit1.Em2.ControlNodes".SemiAutuSplice."step".transition[1421] )
      { S7_Templates := "time_type := Time" } #statTonTimer[1421].TON(pt := #SeqDelayTime, et =>)
      Move(in := #JOB_14_STEP_23, out1 => "Unit1.Em2.ControlNodes".SemiAutuSplice.sequence.status.nextStep)
   END_RUNG
   // the same network as SCL:
   #_w1 := ("Unit1.Em2.ControlNodes".SemiAutuSplice.sequence.status.currentStep = #JOB_14_STEP_21) AND "Unit1.Em2.ControlNodes".SemiAutuSplice.sequence.status.seqActive;
   "Unit1.Em2.ControlNodes".SemiAutuSplice."step".action[1421] := #_w1 AND NOT "Unit1.Em2.ControlNodes".cmSupportUnitTransferFwdBwd.monitoring.inWorkPos;
   "Unit1.Em2.ControlNodes".SemiAutuSplice."step".transition[1421] := #_w1 AND "Unit1.Em2.ControlNodes".cmSupportUnitTransferFwdBwd.monitoring.inWorkPos;
   #statTonTimer[1421].TON(IN := #_w1 AND "Unit1.Em2.ControlNodes".SemiAutuSplice."step".transition[1421],
                           PT := #SeqDelayTime);
   IF #statTonTimer[1421].Q THEN
       "Unit1.Em2.ControlNodes".SemiAutuSplice.sequence.status.nextStep := #JOB_14_STEP_23;
   END_IF;
END_REGION

REGION Network 72: Step[1423] : FrameCover WorkPos Command
   RUNG wire#powerrail
      { S7_Templates := "SrcType := DInt" } EQ_Contact(in1 := "Unit1.Em2.ControlNodes".SemiAutuSplice.sequence.status.currentStep, in2 := #JOB_14_STEP_23)
      Contact( "Unit1.Em2.ControlNodes".SemiAutuSplice.sequence.status.seqActive )
      wire#w1
      I_Contact( "Unit1.Em2.ControlNodes".cmFrameCoverFwdBwd.monitoring.inWorkPos )
      Coil( "Unit1.Em2.ControlNodes".SemiAutuSplice."step".action[1423] )
   END_RUNG
   RUNG wire#w1
      Contact( "Unit1.Em2.ControlNodes".cmFrameCoverFwdBwd.monitoring.inWorkPos )
      Coil( "Unit1.Em2.ControlNodes".SemiAutuSplice."step".transition[1423] )
   END_RUNG
   RUNG wire#w1
      Contact( "Unit1.Em2.ControlNodes".SemiAutuSplice."step".transition[1423] )
      { S7_Templates := "time_type := Time" } #statTonTimer[1423].TON(pt := #SeqDelayTime, et =>)
      Move(in := #JOB_14_STEP_31, out1 => "Unit1.Em2.ControlNodes".SemiAutuSplice.sequence.status.nextStep)
   END_RUNG
   // the same network as SCL:
   #_w1 := ("Unit1.Em2.ControlNodes".SemiAutuSplice.sequence.status.currentStep = #JOB_14_STEP_23) AND "Unit1.Em2.ControlNodes".SemiAutuSplice.sequence.status.seqActive;
   "Unit1.Em2.ControlNodes".SemiAutuSplice."step".action[1423] := #_w1 AND NOT "Unit1.Em2.ControlNodes".cmFrameCoverFwdBwd.monitoring.inWorkPos;
   "Unit1.Em2.ControlNodes".SemiAutuSplice."step".transition[1423] := #_w1 AND "Unit1.Em2.ControlNodes".cmFrameCoverFwdBwd.monitoring.inWorkPos;
   #statTonTimer[1423].TON(IN := #_w1 AND "Unit1.Em2.ControlNodes".SemiAutuSplice."step".transition[1423],
                           PT := #SeqDelayTime);
   IF #statTonTimer[1423].Q THEN
       "Unit1.Em2.ControlNodes".SemiAutuSplice.sequence.status.nextStep := #JOB_14_STEP_31;
   END_IF;
END_REGION

REGION Network 73: Step[1431] : Support Unit Shaft WorkPos Command
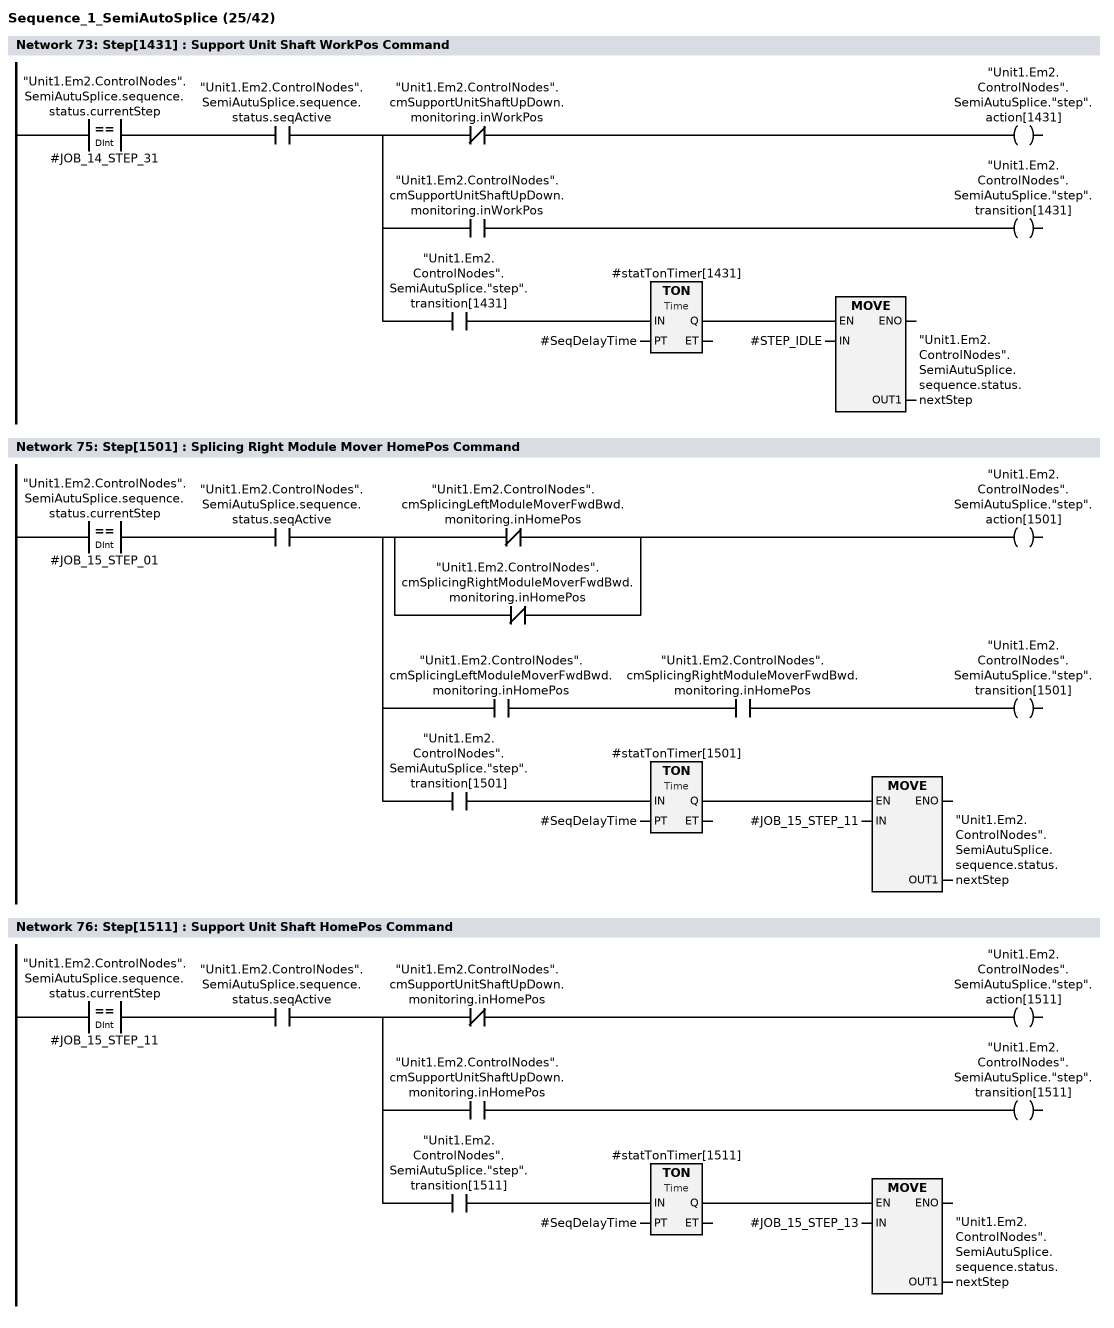
   RUNG wire#powerrail
      { S7_Templates := "SrcType := DInt" } EQ_Contact(in1 := "Unit1.Em2.ControlNodes".SemiAutuSplice.sequence.status.currentStep, in2 := #JOB_14_STEP_31)
      Contact( "Unit1.Em2.ControlNodes".SemiAutuSplice.sequence.status.seqActive )
      wire#w1
      I_Contact( "Unit1.Em2.ControlNodes".cmSupportUnitShaftUpDown.monitoring.inWorkPos )
      Coil( "Unit1.Em2.ControlNodes".SemiAutuSplice."step".action[1431] )
   END_RUNG
   RUNG wire#w1
      Contact( "Unit1.Em2.ControlNodes".cmSupportUnitShaftUpDown.monitoring.inWorkPos )
      Coil( "Unit1.Em2.ControlNodes".SemiAutuSplice."step".transition[1431] )
   END_RUNG
   RUNG wire#w1
      Contact( "Unit1.Em2.ControlNodes".SemiAutuSplice."step".transition[1431] )
      { S7_Templates := "time_type := Time" } #statTonTimer[1431].TON(pt := #SeqDelayTime, et =>)
      Move(in := #STEP_IDLE, out1 => "Unit1.Em2.ControlNodes".SemiAutuSplice.sequence.status.nextStep)
   END_RUNG
   // the same network as SCL:
   #_w1 := ("Unit1.Em2.ControlNodes".SemiAutuSplice.sequence.status.currentStep = #JOB_14_STEP_31) AND "Unit1.Em2.ControlNodes".SemiAutuSplice.sequence.status.seqActive;
   "Unit1.Em2.ControlNodes".SemiAutuSplice."step".action[1431] := #_w1 AND NOT "Unit1.Em2.ControlNodes".cmSupportUnitShaftUpDown.monitoring.inWorkPos;
   "Unit1.Em2.ControlNodes".SemiAutuSplice."step".transition[1431] := #_w1 AND "Unit1.Em2.ControlNodes".cmSupportUnitShaftUpDown.monitoring.inWorkPos;
   #statTonTimer[1431].TON(IN := #_w1 AND "Unit1.Em2.ControlNodes".SemiAutuSplice."step".transition[1431],
                           PT := #SeqDelayTime);
   IF #statTonTimer[1431].Q THEN
       "Unit1.Em2.ControlNodes".SemiAutuSplice.sequence.status.nextStep := #STEP_IDLE;
   END_IF;
END_REGION

REGION Network 74: ******************** JOB[15] RIGHT SPLICING MODULE MOVER AUTO ********************
END_REGION

REGION Network 75: Step[1501] : Splicing Right Module Mover HomePos Command
   RUNG wire#powerrail
      { S7_Templates := "SrcType := DInt" } EQ_Contact(in1 := "Unit1.Em2.ControlNodes".SemiAutuSplice.sequence.status.currentStep, in2 := #JOB_15_STEP_01)
      Contact( "Unit1.Em2.ControlNodes".SemiAutuSplice.sequence.status.seqActive )
      wire#w1
      I_Contact( "Unit1.Em2.ControlNodes".cmSplicingLeftModuleMoverFwdBwd.monitoring.inHomePos )
      wire#w2
      Coil( "Unit1.Em2.ControlNodes".SemiAutuSplice."step".action[1501] )
   END_RUNG
   RUNG wire#w1
      I_Contact( "Unit1.Em2.ControlNodes".cmSplicingRightModuleMoverFwdBwd.monitoring.inHomePos )
   END_RUNG wire#w2
   RUNG wire#w1
      Contact( "Unit1.Em2.ControlNodes".cmSplicingLeftModuleMoverFwdBwd.monitoring.inHomePos )
      Contact( "Unit1.Em2.ControlNodes".cmSplicingRightModuleMoverFwdBwd.monitoring.inHomePos )
      Coil( "Unit1.Em2.ControlNodes".SemiAutuSplice."step".transition[1501] )
   END_RUNG
   RUNG wire#w1
      Contact( "Unit1.Em2.ControlNodes".SemiAutuSplice."step".transition[1501] )
      { S7_Templates := "time_type := Time" } #statTonTimer[1501].TON(pt := #SeqDelayTime, et =>)
      Move(in := #JOB_15_STEP_11, out1 => "Unit1.Em2.ControlNodes".SemiAutuSplice.sequence.status.nextStep)
   END_RUNG
   // the same network as SCL:
   #_w1 := ("Unit1.Em2.ControlNodes".SemiAutuSplice.sequence.status.currentStep = #JOB_15_STEP_01) AND "Unit1.Em2.ControlNodes".SemiAutuSplice.sequence.status.seqActive;
   "Unit1.Em2.ControlNodes".SemiAutuSplice."step".action[1501] := #_w1 AND (NOT "Unit1.Em2.ControlNodes".cmSplicingLeftModuleMoverFwdBwd.monitoring.inHomePos OR NOT "Unit1.Em2.ControlNodes".cmSplicingRightModuleMoverFwdBwd.monitoring.inHomePos);
   "Unit1.Em2.ControlNodes".SemiAutuSplice."step".transition[1501] := #_w1 AND "Unit1.Em2.ControlNodes".cmSplicingLeftModuleMoverFwdBwd.monitoring.inHomePos AND "Unit1.Em2.ControlNodes".cmSplicingRightModuleMoverFwdBwd.monitoring.inHomePos;
   #statTonTimer[1501].TON(IN := #_w1 AND "Unit1.Em2.ControlNodes".SemiAutuSplice."step".transition[1501],
                           PT := #SeqDelayTime);
   IF #statTonTimer[1501].Q THEN
       "Unit1.Em2.ControlNodes".SemiAutuSplice.sequence.status.nextStep := #JOB_15_STEP_11;
   END_IF;
END_REGION

REGION Network 76: Step[1511] : Support Unit Shaft HomePos Command
   RUNG wire#powerrail
      { S7_Templates := "SrcType := DInt" } EQ_Contact(in1 := "Unit1.Em2.ControlNodes".SemiAutuSplice.sequence.status.currentStep, in2 := #JOB_15_STEP_11)
      Contact( "Unit1.Em2.ControlNodes".SemiAutuSplice.sequence.status.seqActive )
      wire#w1
      I_Contact( "Unit1.Em2.ControlNodes".cmSupportUnitShaftUpDown.monitoring.inHomePos )
      Coil( "Unit1.Em2.ControlNodes".SemiAutuSplice."step".action[1511] )
   END_RUNG
   RUNG wire#w1
      Contact( "Unit1.Em2.ControlNodes".cmSupportUnitShaftUpDown.monitoring.inHomePos )
      Coil( "Unit1.Em2.ControlNodes".SemiAutuSplice."step".transition[1511] )
   END_RUNG
   RUNG wire#w1
      Contact( "Unit1.Em2.ControlNodes".SemiAutuSplice."step".transition[1511] )
      { S7_Templates := "time_type := Time" } #statTonTimer[1511].TON(pt := #SeqDelayTime, et =>)
      Move(in := #JOB_15_STEP_13, out1 => "Unit1.Em2.ControlNodes".SemiAutuSplice.sequence.status.nextStep)
   END_RUNG
   // the same network as SCL:
   #_w1 := ("Unit1.Em2.ControlNodes".SemiAutuSplice.sequence.status.currentStep = #JOB_15_STEP_11) AND "Unit1.Em2.ControlNodes".SemiAutuSplice.sequence.status.seqActive;
   "Unit1.Em2.ControlNodes".SemiAutuSplice."step".action[1511] := #_w1 AND NOT "Unit1.Em2.ControlNodes".cmSupportUnitShaftUpDown.monitoring.inHomePos;
   "Unit1.Em2.ControlNodes".SemiAutuSplice."step".transition[1511] := #_w1 AND "Unit1.Em2.ControlNodes".cmSupportUnitShaftUpDown.monitoring.inHomePos;
   #statTonTimer[1511].TON(IN := #_w1 AND "Unit1.Em2.ControlNodes".SemiAutuSplice."step".transition[1511],
                           PT := #SeqDelayTime);
   IF #statTonTimer[1511].Q THEN
       "Unit1.Em2.ControlNodes".SemiAutuSplice.sequence.status.nextStep := #JOB_15_STEP_13;
   END_IF;
END_REGION

REGION Network 77: Step[1513] : FrameCover HomePos Command
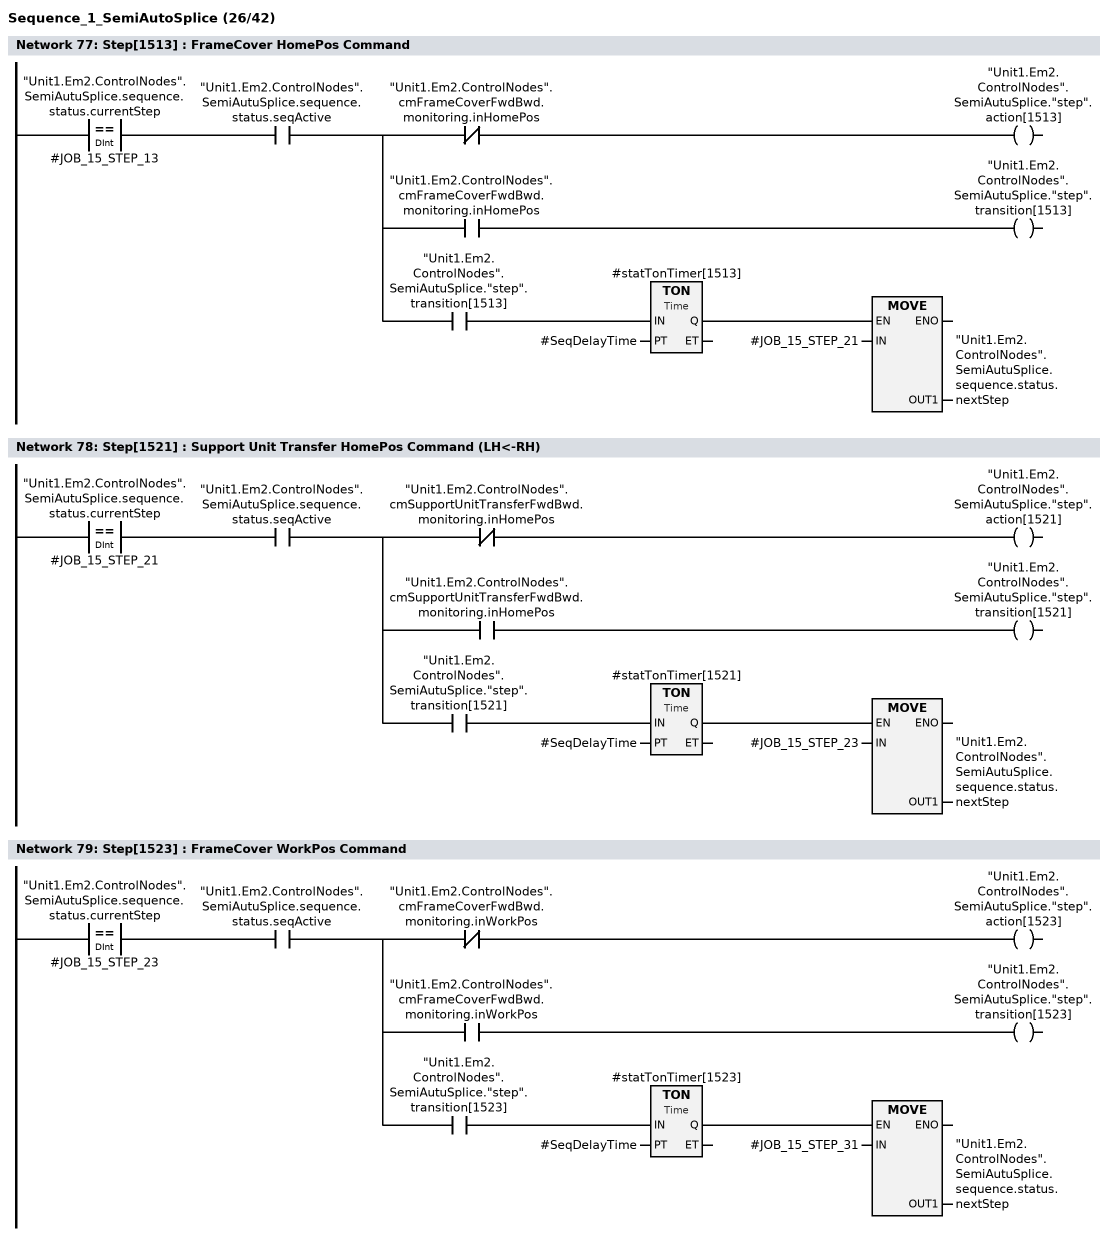
   RUNG wire#powerrail
      { S7_Templates := "SrcType := DInt" } EQ_Contact(in1 := "Unit1.Em2.ControlNodes".SemiAutuSplice.sequence.status.currentStep, in2 := #JOB_15_STEP_13)
      Contact( "Unit1.Em2.ControlNodes".SemiAutuSplice.sequence.status.seqActive )
      wire#w1
      I_Contact( "Unit1.Em2.ControlNodes".cmFrameCoverFwdBwd.monitoring.inHomePos )
      Coil( "Unit1.Em2.ControlNodes".SemiAutuSplice."step".action[1513] )
   END_RUNG
   RUNG wire#w1
      Contact( "Unit1.Em2.ControlNodes".cmFrameCoverFwdBwd.monitoring.inHomePos )
      Coil( "Unit1.Em2.ControlNodes".SemiAutuSplice."step".transition[1513] )
   END_RUNG
   RUNG wire#w1
      Contact( "Unit1.Em2.ControlNodes".SemiAutuSplice."step".transition[1513] )
      { S7_Templates := "time_type := Time" } #statTonTimer[1513].TON(pt := #SeqDelayTime, et =>)
      Move(in := #JOB_15_STEP_21, out1 => "Unit1.Em2.ControlNodes".SemiAutuSplice.sequence.status.nextStep)
   END_RUNG
   // the same network as SCL:
   #_w1 := ("Unit1.Em2.ControlNodes".SemiAutuSplice.sequence.status.currentStep = #JOB_15_STEP_13) AND "Unit1.Em2.ControlNodes".SemiAutuSplice.sequence.status.seqActive;
   "Unit1.Em2.ControlNodes".SemiAutuSplice."step".action[1513] := #_w1 AND NOT "Unit1.Em2.ControlNodes".cmFrameCoverFwdBwd.monitoring.inHomePos;
   "Unit1.Em2.ControlNodes".SemiAutuSplice."step".transition[1513] := #_w1 AND "Unit1.Em2.ControlNodes".cmFrameCoverFwdBwd.monitoring.inHomePos;
   #statTonTimer[1513].TON(IN := #_w1 AND "Unit1.Em2.ControlNodes".SemiAutuSplice."step".transition[1513],
                           PT := #SeqDelayTime);
   IF #statTonTimer[1513].Q THEN
       "Unit1.Em2.ControlNodes".SemiAutuSplice.sequence.status.nextStep := #JOB_15_STEP_21;
   END_IF;
END_REGION

REGION Network 78: Step[1521] : Support Unit Transfer HomePos Command (LH<-RH)
   RUNG wire#powerrail
      { S7_Templates := "SrcType := DInt" } EQ_Contact(in1 := "Unit1.Em2.ControlNodes".SemiAutuSplice.sequence.status.currentStep, in2 := #JOB_15_STEP_21)
      Contact( "Unit1.Em2.ControlNodes".SemiAutuSplice.sequence.status.seqActive )
      wire#w1
      I_Contact( "Unit1.Em2.ControlNodes".cmSupportUnitTransferFwdBwd.monitoring.inHomePos )
      Coil( "Unit1.Em2.ControlNodes".SemiAutuSplice."step".action[1521] )
   END_RUNG
   RUNG wire#w1
      Contact( "Unit1.Em2.ControlNodes".cmSupportUnitTransferFwdBwd.monitoring.inHomePos )
      Coil( "Unit1.Em2.ControlNodes".SemiAutuSplice."step".transition[1521] )
   END_RUNG
   RUNG wire#w1
      Contact( "Unit1.Em2.ControlNodes".SemiAutuSplice."step".transition[1521] )
      { S7_Templates := "time_type := Time" } #statTonTimer[1521].TON(pt := #SeqDelayTime, et =>)
      Move(in := #JOB_15_STEP_23, out1 => "Unit1.Em2.ControlNodes".SemiAutuSplice.sequence.status.nextStep)
   END_RUNG
   // the same network as SCL:
   #_w1 := ("Unit1.Em2.ControlNodes".SemiAutuSplice.sequence.status.currentStep = #JOB_15_STEP_21) AND "Unit1.Em2.ControlNodes".SemiAutuSplice.sequence.status.seqActive;
   "Unit1.Em2.ControlNodes".SemiAutuSplice."step".action[1521] := #_w1 AND NOT "Unit1.Em2.ControlNodes".cmSupportUnitTransferFwdBwd.monitoring.inHomePos;
   "Unit1.Em2.ControlNodes".SemiAutuSplice."step".transition[1521] := #_w1 AND "Unit1.Em2.ControlNodes".cmSupportUnitTransferFwdBwd.monitoring.inHomePos;
   #statTonTimer[1521].TON(IN := #_w1 AND "Unit1.Em2.ControlNodes".SemiAutuSplice."step".transition[1521],
                           PT := #SeqDelayTime);
   IF #statTonTimer[1521].Q THEN
       "Unit1.Em2.ControlNodes".SemiAutuSplice.sequence.status.nextStep := #JOB_15_STEP_23;
   END_IF;
END_REGION

REGION Network 79: Step[1523] : FrameCover WorkPos Command
   RUNG wire#powerrail
      { S7_Templates := "SrcType := DInt" } EQ_Contact(in1 := "Unit1.Em2.ControlNodes".SemiAutuSplice.sequence.status.currentStep, in2 := #JOB_15_STEP_23)
      Contact( "Unit1.Em2.ControlNodes".SemiAutuSplice.sequence.status.seqActive )
      wire#w1
      I_Contact( "Unit1.Em2.ControlNodes".cmFrameCoverFwdBwd.monitoring.inWorkPos )
      Coil( "Unit1.Em2.ControlNodes".SemiAutuSplice."step".action[1523] )
   END_RUNG
   RUNG wire#w1
      Contact( "Unit1.Em2.ControlNodes".cmFrameCoverFwdBwd.monitoring.inWorkPos )
      Coil( "Unit1.Em2.ControlNodes".SemiAutuSplice."step".transition[1523] )
   END_RUNG
   RUNG wire#w1
      Contact( "Unit1.Em2.ControlNodes".SemiAutuSplice."step".transition[1523] )
      { S7_Templates := "time_type := Time" } #statTonTimer[1523].TON(pt := #SeqDelayTime, et =>)
      Move(in := #JOB_15_STEP_31, out1 => "Unit1.Em2.ControlNodes".SemiAutuSplice.sequence.status.nextStep)
   END_RUNG
   // the same network as SCL:
   #_w1 := ("Unit1.Em2.ControlNodes".SemiAutuSplice.sequence.status.currentStep = #JOB_15_STEP_23) AND "Unit1.Em2.ControlNodes".SemiAutuSplice.sequence.status.seqActive;
   "Unit1.Em2.ControlNodes".SemiAutuSplice."step".action[1523] := #_w1 AND NOT "Unit1.Em2.ControlNodes".cmFrameCoverFwdBwd.monitoring.inWorkPos;
   "Unit1.Em2.ControlNodes".SemiAutuSplice."step".transition[1523] := #_w1 AND "Unit1.Em2.ControlNodes".cmFrameCoverFwdBwd.monitoring.inWorkPos;
   #statTonTimer[1523].TON(IN := #_w1 AND "Unit1.Em2.ControlNodes".SemiAutuSplice."step".transition[1523],
                           PT := #SeqDelayTime);
   IF #statTonTimer[1523].Q THEN
       "Unit1.Em2.ControlNodes".SemiAutuSplice.sequence.status.nextStep := #JOB_15_STEP_31;
   END_IF;
END_REGION

REGION Network 80: Step[1531] : Support Unit Shaft WorkPos Command
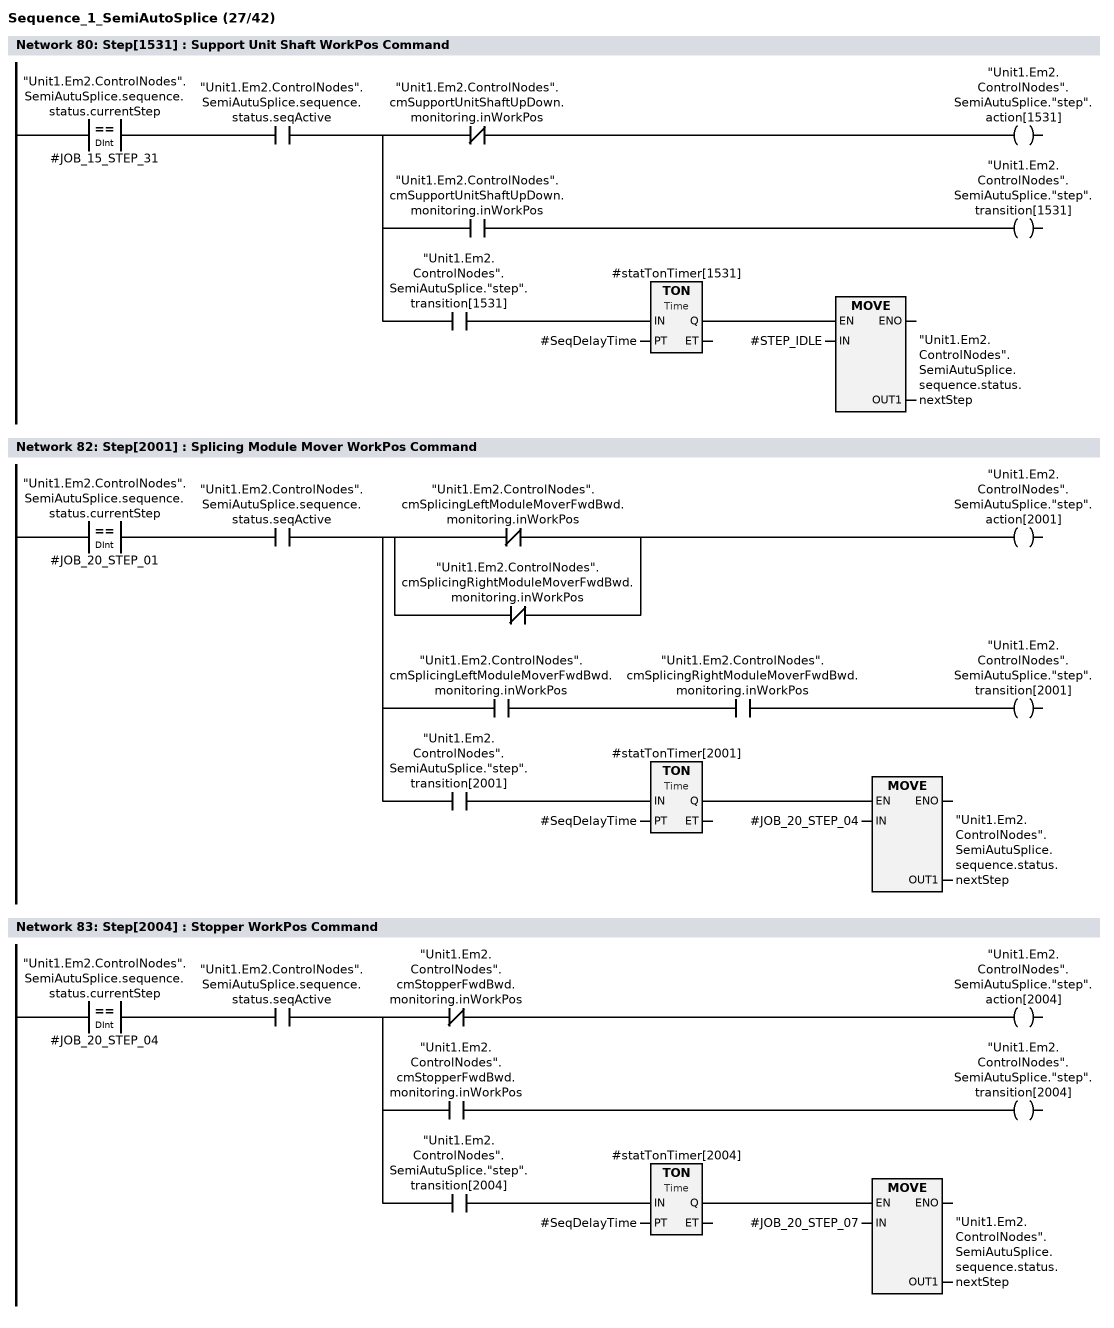
   RUNG wire#powerrail
      { S7_Templates := "SrcType := DInt" } EQ_Contact(in1 := "Unit1.Em2.ControlNodes".SemiAutuSplice.sequence.status.currentStep, in2 := #JOB_15_STEP_31)
      Contact( "Unit1.Em2.ControlNodes".SemiAutuSplice.sequence.status.seqActive )
      wire#w1
      I_Contact( "Unit1.Em2.ControlNodes".cmSupportUnitShaftUpDown.monitoring.inWorkPos )
      Coil( "Unit1.Em2.ControlNodes".SemiAutuSplice."step".action[1531] )
   END_RUNG
   RUNG wire#w1
      Contact( "Unit1.Em2.ControlNodes".cmSupportUnitShaftUpDown.monitoring.inWorkPos )
      Coil( "Unit1.Em2.ControlNodes".SemiAutuSplice."step".transition[1531] )
   END_RUNG
   RUNG wire#w1
      Contact( "Unit1.Em2.ControlNodes".SemiAutuSplice."step".transition[1531] )
      { S7_Templates := "time_type := Time" } #statTonTimer[1531].TON(pt := #SeqDelayTime, et =>)
      Move(in := #STEP_IDLE, out1 => "Unit1.Em2.ControlNodes".SemiAutuSplice.sequence.status.nextStep)
   END_RUNG
   // the same network as SCL:
   #_w1 := ("Unit1.Em2.ControlNodes".SemiAutuSplice.sequence.status.currentStep = #JOB_15_STEP_31) AND "Unit1.Em2.ControlNodes".SemiAutuSplice.sequence.status.seqActive;
   "Unit1.Em2.ControlNodes".SemiAutuSplice."step".action[1531] := #_w1 AND NOT "Unit1.Em2.ControlNodes".cmSupportUnitShaftUpDown.monitoring.inWorkPos;
   "Unit1.Em2.ControlNodes".SemiAutuSplice."step".transition[1531] := #_w1 AND "Unit1.Em2.ControlNodes".cmSupportUnitShaftUpDown.monitoring.inWorkPos;
   #statTonTimer[1531].TON(IN := #_w1 AND "Unit1.Em2.ControlNodes".SemiAutuSplice."step".transition[1531],
                           PT := #SeqDelayTime);
   IF #statTonTimer[1531].Q THEN
       "Unit1.Em2.ControlNodes".SemiAutuSplice.sequence.status.nextStep := #STEP_IDLE;
   END_IF;
END_REGION

REGION Network 81: ******************** JOB[20] FULL AUTO SPLICING ********************
END_REGION

REGION Network 82: Step[2001] : Splicing Module Mover WorkPos Command
   RUNG wire#powerrail
      { S7_Templates := "SrcType := DInt" } EQ_Contact(in1 := "Unit1.Em2.ControlNodes".SemiAutuSplice.sequence.status.currentStep, in2 := #JOB_20_STEP_01)
      Contact( "Unit1.Em2.ControlNodes".SemiAutuSplice.sequence.status.seqActive )
      wire#w1
      I_Contact( "Unit1.Em2.ControlNodes".cmSplicingLeftModuleMoverFwdBwd.monitoring.inWorkPos )
      wire#w2
      Coil( "Unit1.Em2.ControlNodes".SemiAutuSplice."step".action[2001] )
   END_RUNG
   RUNG wire#w1
      I_Contact( "Unit1.Em2.ControlNodes".cmSplicingRightModuleMoverFwdBwd.monitoring.inWorkPos )
   END_RUNG wire#w2
   RUNG wire#w1
      Contact( "Unit1.Em2.ControlNodes".cmSplicingLeftModuleMoverFwdBwd.monitoring.inWorkPos )
      Contact( "Unit1.Em2.ControlNodes".cmSplicingRightModuleMoverFwdBwd.monitoring.inWorkPos )
      Coil( "Unit1.Em2.ControlNodes".SemiAutuSplice."step".transition[2001] )
   END_RUNG
   RUNG wire#w1
      Contact( "Unit1.Em2.ControlNodes".SemiAutuSplice."step".transition[2001] )
      { S7_Templates := "time_type := Time" } #statTonTimer[2001].TON(pt := #SeqDelayTime, et =>)
      Move(in := #JOB_20_STEP_04, out1 => "Unit1.Em2.ControlNodes".SemiAutuSplice.sequence.status.nextStep)
   END_RUNG
   // the same network as SCL:
   #_w1 := ("Unit1.Em2.ControlNodes".SemiAutuSplice.sequence.status.currentStep = #JOB_20_STEP_01) AND "Unit1.Em2.ControlNodes".SemiAutuSplice.sequence.status.seqActive;
   "Unit1.Em2.ControlNodes".SemiAutuSplice."step".action[2001] := #_w1 AND (NOT "Unit1.Em2.ControlNodes".cmSplicingLeftModuleMoverFwdBwd.monitoring.inWorkPos OR NOT "Unit1.Em2.ControlNodes".cmSplicingRightModuleMoverFwdBwd.monitoring.inWorkPos);
   "Unit1.Em2.ControlNodes".SemiAutuSplice."step".transition[2001] := #_w1 AND "Unit1.Em2.ControlNodes".cmSplicingLeftModuleMoverFwdBwd.monitoring.inWorkPos AND "Unit1.Em2.ControlNodes".cmSplicingRightModuleMoverFwdBwd.monitoring.inWorkPos;
   #statTonTimer[2001].TON(IN := #_w1 AND "Unit1.Em2.ControlNodes".SemiAutuSplice."step".transition[2001],
                           PT := #SeqDelayTime);
   IF #statTonTimer[2001].Q THEN
       "Unit1.Em2.ControlNodes".SemiAutuSplice.sequence.status.nextStep := #JOB_20_STEP_04;
   END_IF;
END_REGION

REGION Network 83: Step[2004] : Stopper WorkPos Command
   RUNG wire#powerrail
      { S7_Templates := "SrcType := DInt" } EQ_Contact(in1 := "Unit1.Em2.ControlNodes".SemiAutuSplice.sequence.status.currentStep, in2 := #JOB_20_STEP_04)
      Contact( "Unit1.Em2.ControlNodes".SemiAutuSplice.sequence.status.seqActive )
      wire#w1
      I_Contact( "Unit1.Em2.ControlNodes".cmStopperFwdBwd.monitoring.inWorkPos )
      Coil( "Unit1.Em2.ControlNodes".SemiAutuSplice."step".action[2004] )
   END_RUNG
   RUNG wire#w1
      Contact( "Unit1.Em2.ControlNodes".cmStopperFwdBwd.monitoring.inWorkPos )
      Coil( "Unit1.Em2.ControlNodes".SemiAutuSplice."step".transition[2004] )
   END_RUNG
   RUNG wire#w1
      Contact( "Unit1.Em2.ControlNodes".SemiAutuSplice."step".transition[2004] )
      { S7_Templates := "time_type := Time" } #statTonTimer[2004].TON(pt := #SeqDelayTime, et =>)
      Move(in := #JOB_20_STEP_07, out1 => "Unit1.Em2.ControlNodes".SemiAutuSplice.sequence.status.nextStep)
   END_RUNG
   // the same network as SCL:
   #_w1 := ("Unit1.Em2.ControlNodes".SemiAutuSplice.sequence.status.currentStep = #JOB_20_STEP_04) AND "Unit1.Em2.ControlNodes".SemiAutuSplice.sequence.status.seqActive;
   "Unit1.Em2.ControlNodes".SemiAutuSplice."step".action[2004] := #_w1 AND NOT "Unit1.Em2.ControlNodes".cmStopperFwdBwd.monitoring.inWorkPos;
   "Unit1.Em2.ControlNodes".SemiAutuSplice."step".transition[2004] := #_w1 AND "Unit1.Em2.ControlNodes".cmStopperFwdBwd.monitoring.inWorkPos;
   #statTonTimer[2004].TON(IN := #_w1 AND "Unit1.Em2.ControlNodes".SemiAutuSplice."step".transition[2004],
                           PT := #SeqDelayTime);
   IF #statTonTimer[2004].Q THEN
       "Unit1.Em2.ControlNodes".SemiAutuSplice.sequence.status.nextStep := #JOB_20_STEP_07;
   END_IF;
END_REGION

REGION Network 84: Step[2007] : Electrode Fix Top Down & Electrode Fix Bottom Up WorkPos Command
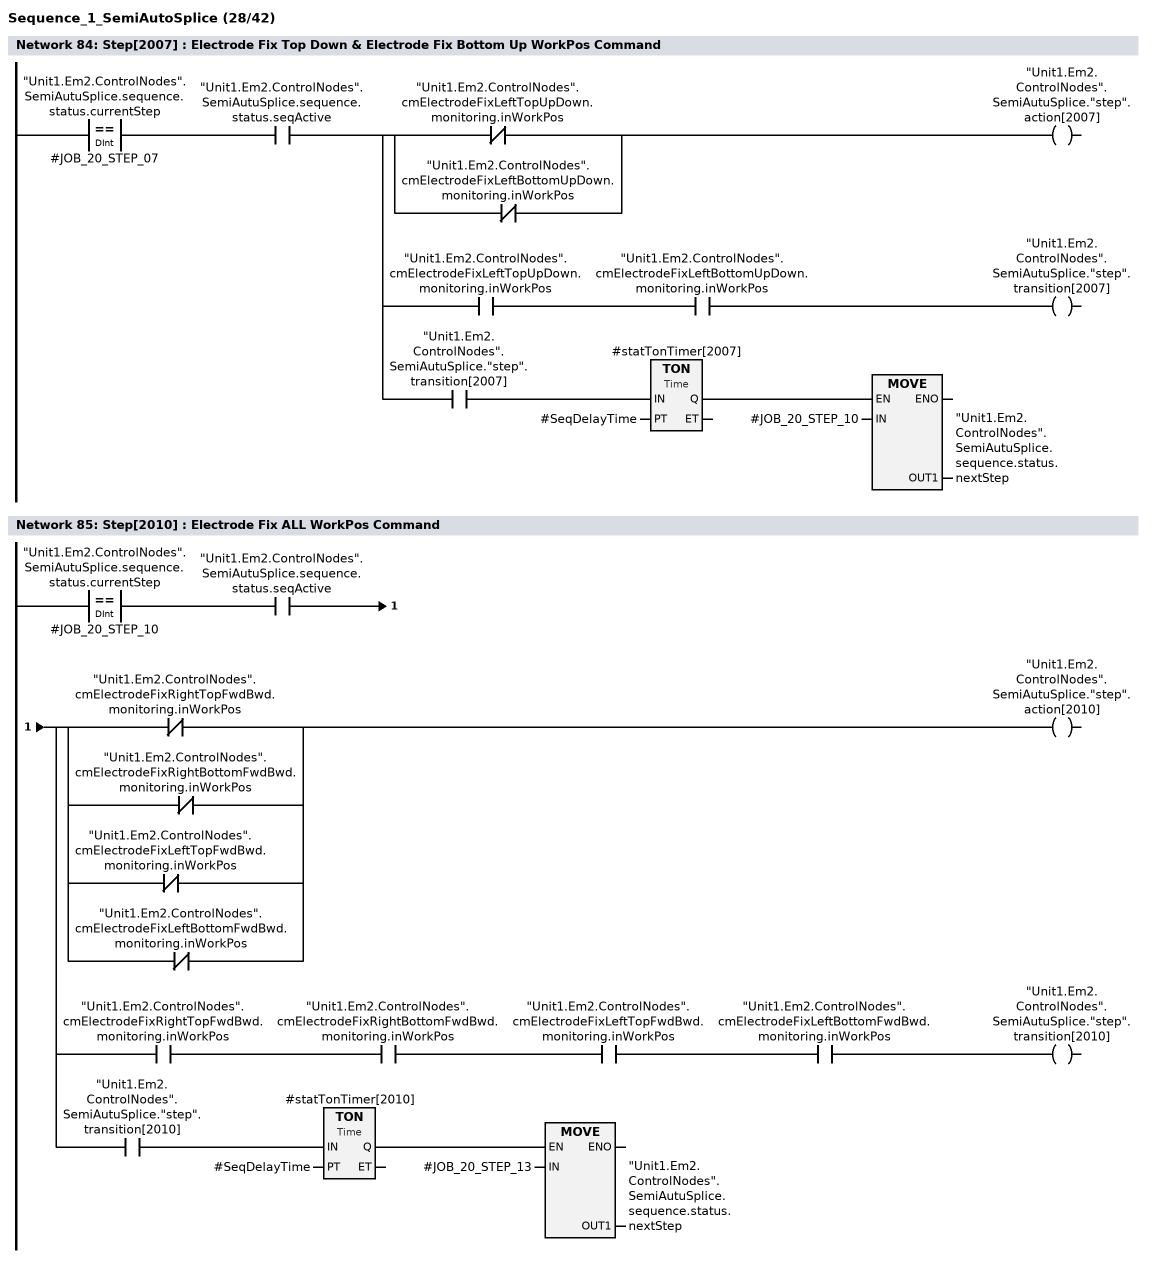
   RUNG wire#powerrail
      { S7_Templates := "SrcType := DInt" } EQ_Contact(in1 := "Unit1.Em2.ControlNodes".SemiAutuSplice.sequence.status.currentStep, in2 := #JOB_20_STEP_07)
      Contact( "Unit1.Em2.ControlNodes".SemiAutuSplice.sequence.status.seqActive )
      wire#w1
      I_Contact( "Unit1.Em2.ControlNodes".cmElectrodeFixLeftTopUpDown.monitoring.inWorkPos )
      wire#w2
      Coil( "Unit1.Em2.ControlNodes".SemiAutuSplice."step".action[2007] )
   END_RUNG
   RUNG wire#w1
      I_Contact( "Unit1.Em2.ControlNodes".cmElectrodeFixLeftBottomUpDown.monitoring.inWorkPos )
   END_RUNG wire#w2
   RUNG wire#w1
      Contact( "Unit1.Em2.ControlNodes".cmElectrodeFixLeftTopUpDown.monitoring.inWorkPos )
      Contact( "Unit1.Em2.ControlNodes".cmElectrodeFixLeftBottomUpDown.monitoring.inWorkPos )
      Coil( "Unit1.Em2.ControlNodes".SemiAutuSplice."step".transition[2007] )
   END_RUNG
   RUNG wire#w1
      Contact( "Unit1.Em2.ControlNodes".SemiAutuSplice."step".transition[2007] )
      { S7_Templates := "time_type := Time" } #statTonTimer[2007].TON(pt := #SeqDelayTime, et =>)
      Move(in := #JOB_20_STEP_10, out1 => "Unit1.Em2.ControlNodes".SemiAutuSplice.sequence.status.nextStep)
   END_RUNG
   // the same network as SCL:
   #_w1 := ("Unit1.Em2.ControlNodes".SemiAutuSplice.sequence.status.currentStep = #JOB_20_STEP_07) AND "Unit1.Em2.ControlNodes".SemiAutuSplice.sequence.status.seqActive;
   "Unit1.Em2.ControlNodes".SemiAutuSplice."step".action[2007] := #_w1 AND (NOT "Unit1.Em2.ControlNodes".cmElectrodeFixLeftTopUpDown.monitoring.inWorkPos OR NOT "Unit1.Em2.ControlNodes".cmElectrodeFixLeftBottomUpDown.monitoring.inWorkPos);
   "Unit1.Em2.ControlNodes".SemiAutuSplice."step".transition[2007] := #_w1 AND "Unit1.Em2.ControlNodes".cmElectrodeFixLeftTopUpDown.monitoring.inWorkPos AND "Unit1.Em2.ControlNodes".cmElectrodeFixLeftBottomUpDown.monitoring.inWorkPos;
   #statTonTimer[2007].TON(IN := #_w1 AND "Unit1.Em2.ControlNodes".SemiAutuSplice."step".transition[2007],
                           PT := #SeqDelayTime);
   IF #statTonTimer[2007].Q THEN
       "Unit1.Em2.ControlNodes".SemiAutuSplice.sequence.status.nextStep := #JOB_20_STEP_10;
   END_IF;
END_REGION

REGION Network 85: Step[2010] : Electrode Fix ALL WorkPos Command
   RUNG wire#powerrail
      { S7_Templates := "SrcType := DInt" } EQ_Contact(in1 := "Unit1.Em2.ControlNodes".SemiAutuSplice.sequence.status.currentStep, in2 := #JOB_20_STEP_10)
      Contact( "Unit1.Em2.ControlNodes".SemiAutuSplice.sequence.status.seqActive )
      wire#w1
      I_Contact( "Unit1.Em2.ControlNodes".cmElectrodeFixRightTopFwdBwd.monitoring.inWorkPos )
      wire#w2
      Coil( "Unit1.Em2.ControlNodes".SemiAutuSplice."step".action[2010] )
   END_RUNG
   RUNG wire#w1
      I_Contact( "Unit1.Em2.ControlNodes".cmElectrodeFixRightBottomFwdBwd.monitoring.inWorkPos )
   END_RUNG wire#w2
   RUNG wire#w1
      I_Contact( "Unit1.Em2.ControlNodes".cmElectrodeFixLeftTopFwdBwd.monitoring.inWorkPos )
   END_RUNG wire#w2
   RUNG wire#w1
      I_Contact( "Unit1.Em2.ControlNodes".cmElectrodeFixLeftBottomFwdBwd.monitoring.inWorkPos )
   END_RUNG wire#w2
   RUNG wire#w1
      Contact( "Unit1.Em2.ControlNodes".cmElectrodeFixRightTopFwdBwd.monitoring.inWorkPos )
      Contact( "Unit1.Em2.ControlNodes".cmElectrodeFixRightBottomFwdBwd.monitoring.inWorkPos )
      Contact( "Unit1.Em2.ControlNodes".cmElectrodeFixLeftTopFwdBwd.monitoring.inWorkPos )
      Contact( "Unit1.Em2.ControlNodes".cmElectrodeFixLeftBottomFwdBwd.monitoring.inWorkPos )
      Coil( "Unit1.Em2.ControlNodes".SemiAutuSplice."step".transition[2010] )
   END_RUNG
   RUNG wire#w1
      Contact( "Unit1.Em2.ControlNodes".SemiAutuSplice."step".transition[2010] )
      { S7_Templates := "time_type := Time" } #statTonTimer[2010].TON(pt := #SeqDelayTime, et =>)
      Move(in := #JOB_20_STEP_13, out1 => "Unit1.Em2.ControlNodes".SemiAutuSplice.sequence.status.nextStep)
   END_RUNG
   // the same network as SCL:
   #_w1 := ("Unit1.Em2.ControlNodes".SemiAutuSplice.sequence.status.currentStep = #JOB_20_STEP_10) AND "Unit1.Em2.ControlNodes".SemiAutuSplice.sequence.status.seqActive;
   "Unit1.Em2.ControlNodes".SemiAutuSplice."step".action[2010] := #_w1 AND (NOT "Unit1.Em2.ControlNodes".cmElectrodeFixRightTopFwdBwd.monitoring.inWorkPos OR NOT "Unit1.Em2.ControlNodes".cmElectrodeFixRightBottomFwdBwd.monitoring.inWorkPos OR NOT "Unit1.Em2.ControlNodes".cmElectrodeFixLeftTopFwdBwd.monitoring.inWorkPos OR NOT "Unit1.Em2.ControlNodes".cmElectrodeFixLeftBottomFwdBwd.monitoring.inWorkPos);
   "Unit1.Em2.ControlNodes".SemiAutuSplice."step".transition[2010] := #_w1 AND "Unit1.Em2.ControlNodes".cmElectrodeFixRightTopFwdBwd.monitoring.inWorkPos AND "Unit1.Em2.ControlNodes".cmElectrodeFixRightBottomFwdBwd.monitoring.inWorkPos AND "Unit1.Em2.ControlNodes".cmElectrodeFixLeftTopFwdBwd.monitoring.inWorkPos AND "Unit1.Em2.ControlNodes".cmElectrodeFixLeftBottomFwdBwd.monitoring.inWorkPos;
   #statTonTimer[2010].TON(IN := #_w1 AND "Unit1.Em2.ControlNodes".SemiAutuSplice."step".transition[2010],
                           PT := #SeqDelayTime);
   IF #statTonTimer[2010].Q THEN
       "Unit1.Em2.ControlNodes".SemiAutuSplice.sequence.status.nextStep := #JOB_20_STEP_13;
   END_IF;
END_REGION

REGION Network 86: Step[2013] : Uw Semi Splicer Vacuum All WorkPos Command
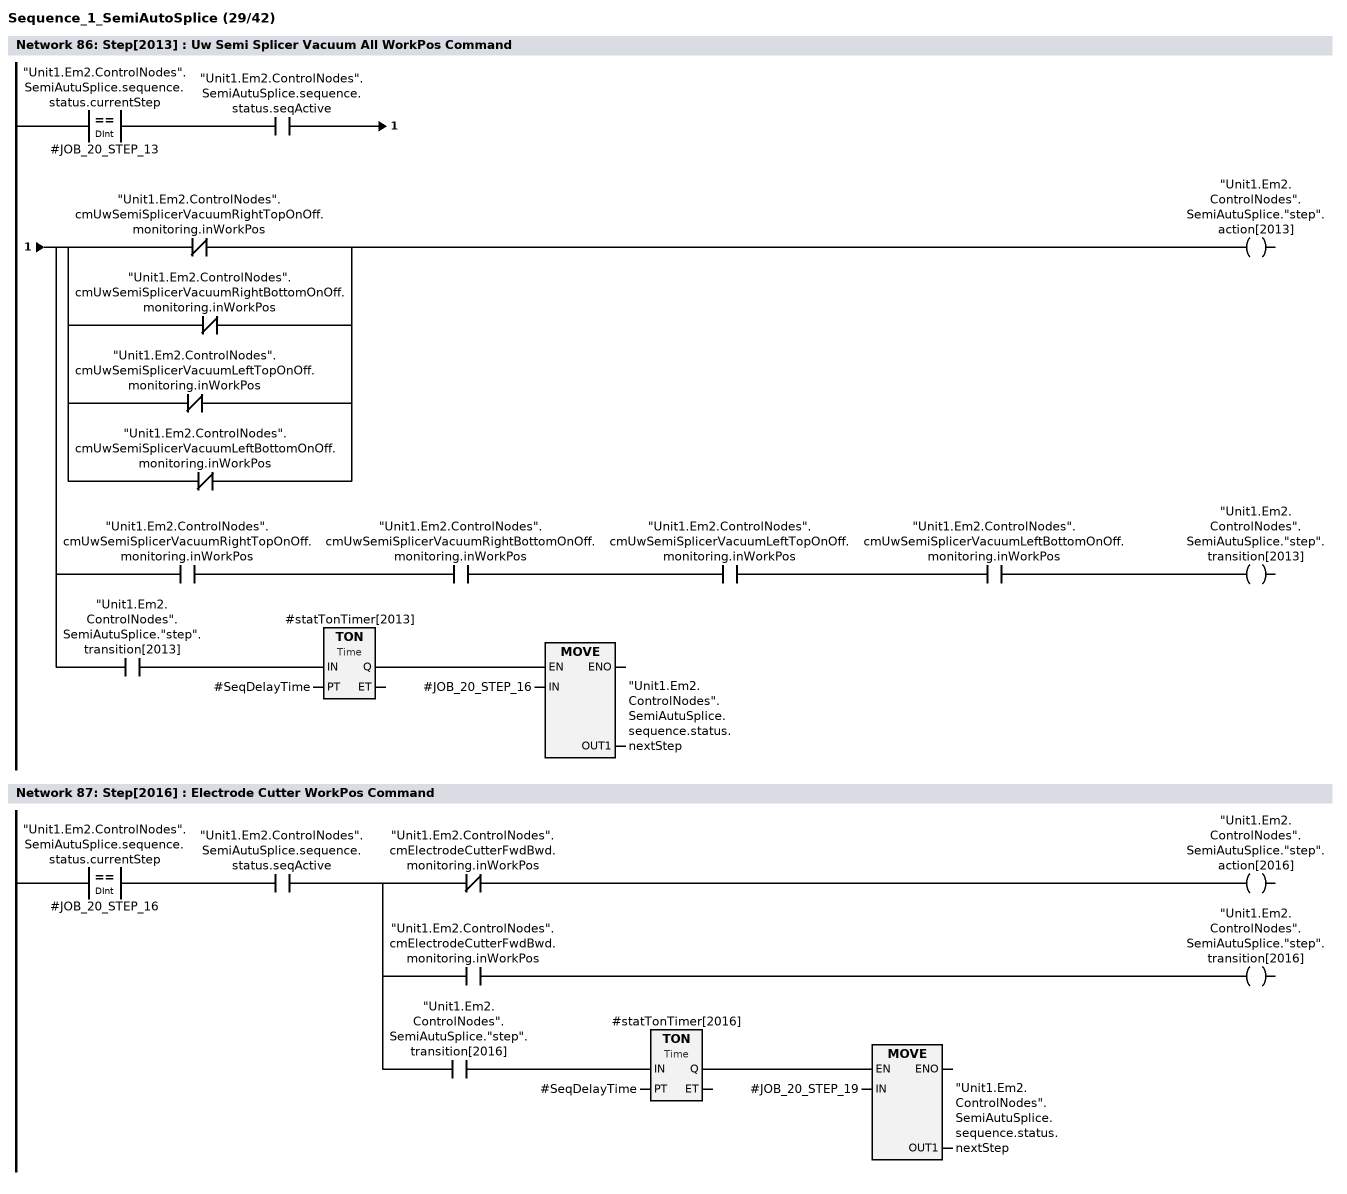
   RUNG wire#powerrail
      { S7_Templates := "SrcType := DInt" } EQ_Contact(in1 := "Unit1.Em2.ControlNodes".SemiAutuSplice.sequence.status.currentStep, in2 := #JOB_20_STEP_13)
      Contact( "Unit1.Em2.ControlNodes".SemiAutuSplice.sequence.status.seqActive )
      wire#w1
      I_Contact( "Unit1.Em2.ControlNodes".cmUwSemiSplicerVacuumRightTopOnOff.monitoring.inWorkPos )
      wire#w2
      Coil( "Unit1.Em2.ControlNodes".SemiAutuSplice."step".action[2013] )
   END_RUNG
   RUNG wire#w1
      I_Contact( "Unit1.Em2.ControlNodes".cmUwSemiSplicerVacuumRightBottomOnOff.monitoring.inWorkPos )
   END_RUNG wire#w2
   RUNG wire#w1
      I_Contact( "Unit1.Em2.ControlNodes".cmUwSemiSplicerVacuumLeftTopOnOff.monitoring.inWorkPos )
   END_RUNG wire#w2
   RUNG wire#w1
      I_Contact( "Unit1.Em2.ControlNodes".cmUwSemiSplicerVacuumLeftBottomOnOff.monitoring.inWorkPos )
   END_RUNG wire#w2
   RUNG wire#w1
      Contact( "Unit1.Em2.ControlNodes".cmUwSemiSplicerVacuumRightTopOnOff.monitoring.inWorkPos )
      Contact( "Unit1.Em2.ControlNodes".cmUwSemiSplicerVacuumRightBottomOnOff.monitoring.inWorkPos )
      Contact( "Unit1.Em2.ControlNodes".cmUwSemiSplicerVacuumLeftTopOnOff.monitoring.inWorkPos )
      Contact( "Unit1.Em2.ControlNodes".cmUwSemiSplicerVacuumLeftBottomOnOff.monitoring.inWorkPos )
      Coil( "Unit1.Em2.ControlNodes".SemiAutuSplice."step".transition[2013] )
   END_RUNG
   RUNG wire#w1
      Contact( "Unit1.Em2.ControlNodes".SemiAutuSplice."step".transition[2013] )
      { S7_Templates := "time_type := Time" } #statTonTimer[2013].TON(pt := #SeqDelayTime, et =>)
      Move(in := #JOB_20_STEP_16, out1 => "Unit1.Em2.ControlNodes".SemiAutuSplice.sequence.status.nextStep)
   END_RUNG
   // the same network as SCL:
   #_w1 := ("Unit1.Em2.ControlNodes".SemiAutuSplice.sequence.status.currentStep = #JOB_20_STEP_13) AND "Unit1.Em2.ControlNodes".SemiAutuSplice.sequence.status.seqActive;
   "Unit1.Em2.ControlNodes".SemiAutuSplice."step".action[2013] := #_w1 AND (NOT "Unit1.Em2.ControlNodes".cmUwSemiSplicerVacuumRightTopOnOff.monitoring.inWorkPos OR NOT "Unit1.Em2.ControlNodes".cmUwSemiSplicerVacuumRightBottomOnOff.monitoring.inWorkPos OR NOT "Unit1.Em2.ControlNodes".cmUwSemiSplicerVacuumLeftTopOnOff.monitoring.inWorkPos OR NOT "Unit1.Em2.ControlNodes".cmUwSemiSplicerVacuumLeftBottomOnOff.monitoring.inWorkPos);
   "Unit1.Em2.ControlNodes".SemiAutuSplice."step".transition[2013] := #_w1 AND "Unit1.Em2.ControlNodes".cmUwSemiSplicerVacuumRightTopOnOff.monitoring.inWorkPos AND "Unit1.Em2.ControlNodes".cmUwSemiSplicerVacuumRightBottomOnOff.monitoring.inWorkPos AND "Unit1.Em2.ControlNodes".cmUwSemiSplicerVacuumLeftTopOnOff.monitoring.inWorkPos AND "Unit1.Em2.ControlNodes".cmUwSemiSplicerVacuumLeftBottomOnOff.monitoring.inWorkPos;
   #statTonTimer[2013].TON(IN := #_w1 AND "Unit1.Em2.ControlNodes".SemiAutuSplice."step".transition[2013],
                           PT := #SeqDelayTime);
   IF #statTonTimer[2013].Q THEN
       "Unit1.Em2.ControlNodes".SemiAutuSplice.sequence.status.nextStep := #JOB_20_STEP_16;
   END_IF;
END_REGION

REGION Network 87: Step[2016] : Electrode Cutter WorkPos Command
   RUNG wire#powerrail
      { S7_Templates := "SrcType := DInt" } EQ_Contact(in1 := "Unit1.Em2.ControlNodes".SemiAutuSplice.sequence.status.currentStep, in2 := #JOB_20_STEP_16)
      Contact( "Unit1.Em2.ControlNodes".SemiAutuSplice.sequence.status.seqActive )
      wire#w1
      I_Contact( "Unit1.Em2.ControlNodes".cmElectrodeCutterFwdBwd.monitoring.inWorkPos )
      Coil( "Unit1.Em2.ControlNodes".SemiAutuSplice."step".action[2016] )
   END_RUNG
   RUNG wire#w1
      Contact( "Unit1.Em2.ControlNodes".cmElectrodeCutterFwdBwd.monitoring.inWorkPos )
      Coil( "Unit1.Em2.ControlNodes".SemiAutuSplice."step".transition[2016] )
   END_RUNG
   RUNG wire#w1
      Contact( "Unit1.Em2.ControlNodes".SemiAutuSplice."step".transition[2016] )
      { S7_Templates := "time_type := Time" } #statTonTimer[2016].TON(pt := #SeqDelayTime, et =>)
      Move(in := #JOB_20_STEP_19, out1 => "Unit1.Em2.ControlNodes".SemiAutuSplice.sequence.status.nextStep)
   END_RUNG
   // the same network as SCL:
   #_w1 := ("Unit1.Em2.ControlNodes".SemiAutuSplice.sequence.status.currentStep = #JOB_20_STEP_16) AND "Unit1.Em2.ControlNodes".SemiAutuSplice.sequence.status.seqActive;
   "Unit1.Em2.ControlNodes".SemiAutuSplice."step".action[2016] := #_w1 AND NOT "Unit1.Em2.ControlNodes".cmElectrodeCutterFwdBwd.monitoring.inWorkPos;
   "Unit1.Em2.ControlNodes".SemiAutuSplice."step".transition[2016] := #_w1 AND "Unit1.Em2.ControlNodes".cmElectrodeCutterFwdBwd.monitoring.inWorkPos;
   #statTonTimer[2016].TON(IN := #_w1 AND "Unit1.Em2.ControlNodes".SemiAutuSplice."step".transition[2016],
                           PT := #SeqDelayTime);
   IF #statTonTimer[2016].Q THEN
       "Unit1.Em2.ControlNodes".SemiAutuSplice.sequence.status.nextStep := #JOB_20_STEP_19;
   END_IF;
END_REGION

REGION Network 88: Step[2019] : Electrode Cutter HomePos Command
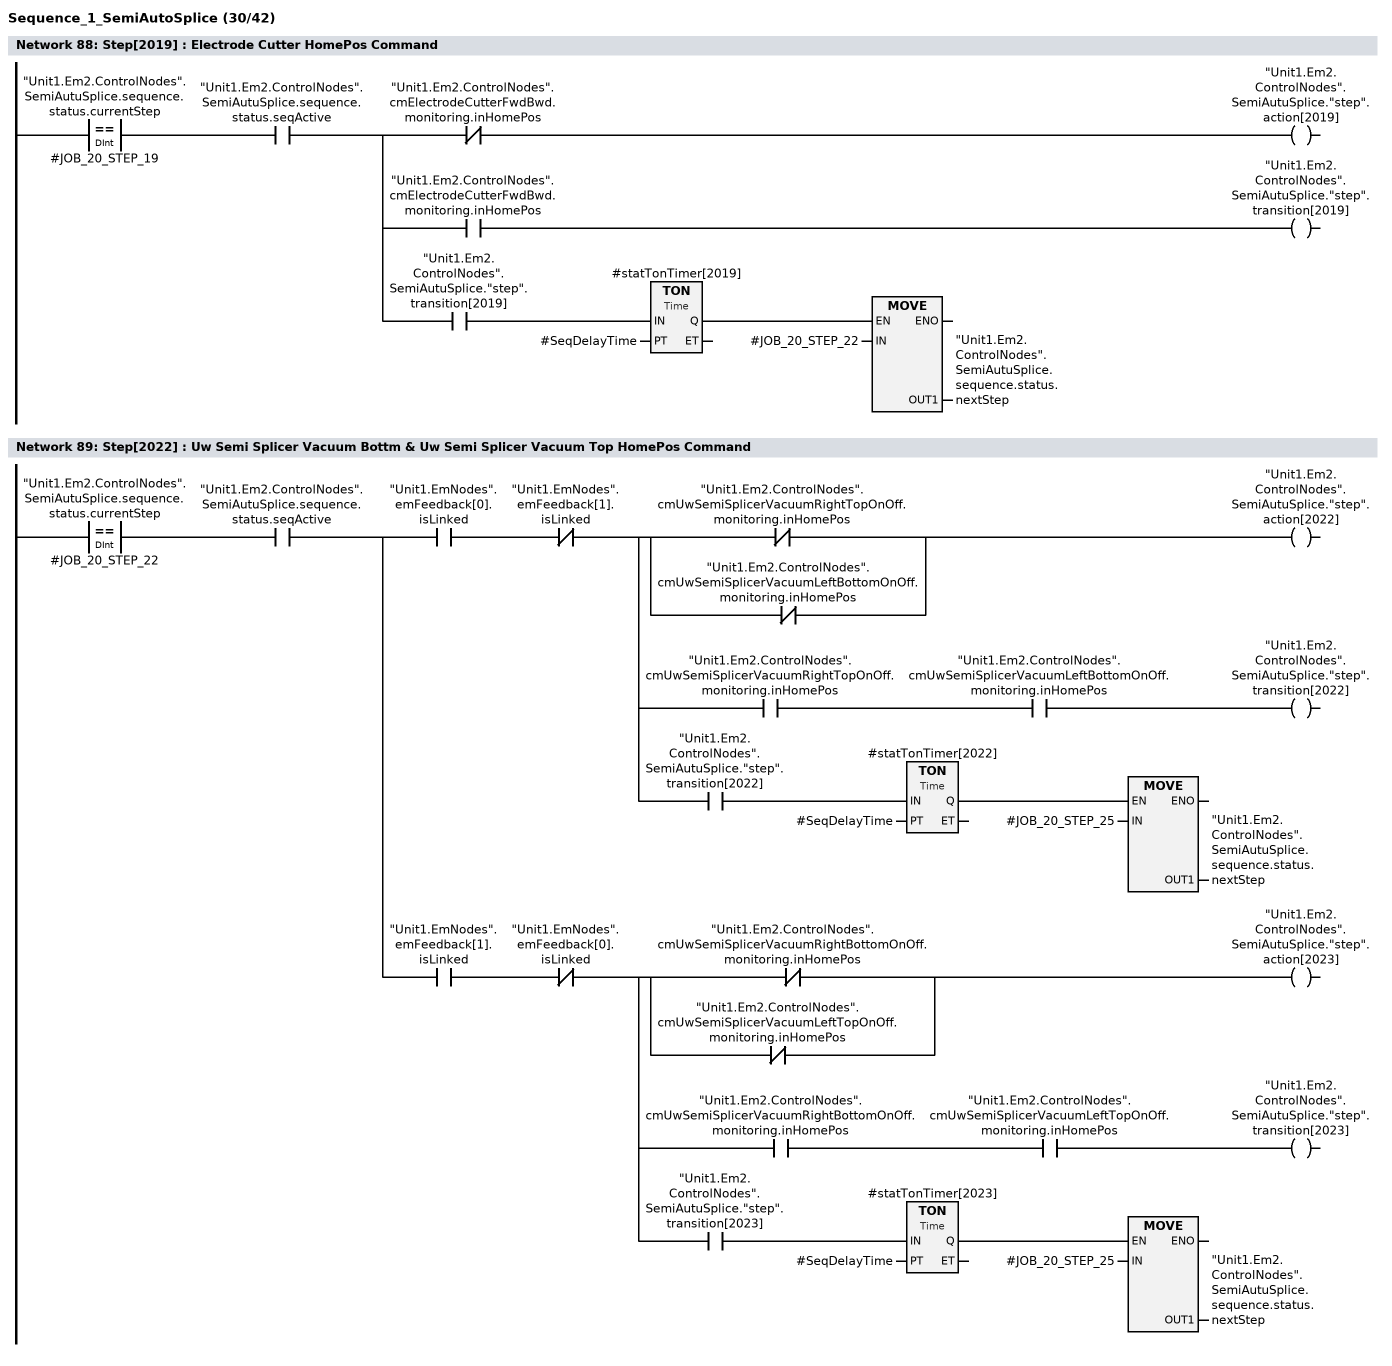
   RUNG wire#powerrail
      { S7_Templates := "SrcType := DInt" } EQ_Contact(in1 := "Unit1.Em2.ControlNodes".SemiAutuSplice.sequence.status.currentStep, in2 := #JOB_20_STEP_19)
      Contact( "Unit1.Em2.ControlNodes".SemiAutuSplice.sequence.status.seqActive )
      wire#w1
      I_Contact( "Unit1.Em2.ControlNodes".cmElectrodeCutterFwdBwd.monitoring.inHomePos )
      Coil( "Unit1.Em2.ControlNodes".SemiAutuSplice."step".action[2019] )
   END_RUNG
   RUNG wire#w1
      Contact( "Unit1.Em2.ControlNodes".cmElectrodeCutterFwdBwd.monitoring.inHomePos )
      Coil( "Unit1.Em2.ControlNodes".SemiAutuSplice."step".transition[2019] )
   END_RUNG
   RUNG wire#w1
      Contact( "Unit1.Em2.ControlNodes".SemiAutuSplice."step".transition[2019] )
      { S7_Templates := "time_type := Time" } #statTonTimer[2019].TON(pt := #SeqDelayTime, et =>)
      Move(in := #JOB_20_STEP_22, out1 => "Unit1.Em2.ControlNodes".SemiAutuSplice.sequence.status.nextStep)
   END_RUNG
   // the same network as SCL:
   #_w1 := ("Unit1.Em2.ControlNodes".SemiAutuSplice.sequence.status.currentStep = #JOB_20_STEP_19) AND "Unit1.Em2.ControlNodes".SemiAutuSplice.sequence.status.seqActive;
   "Unit1.Em2.ControlNodes".SemiAutuSplice."step".action[2019] := #_w1 AND NOT "Unit1.Em2.ControlNodes".cmElectrodeCutterFwdBwd.monitoring.inHomePos;
   "Unit1.Em2.ControlNodes".SemiAutuSplice."step".transition[2019] := #_w1 AND "Unit1.Em2.ControlNodes".cmElectrodeCutterFwdBwd.monitoring.inHomePos;
   #statTonTimer[2019].TON(IN := #_w1 AND "Unit1.Em2.ControlNodes".SemiAutuSplice."step".transition[2019],
                           PT := #SeqDelayTime);
   IF #statTonTimer[2019].Q THEN
       "Unit1.Em2.ControlNodes".SemiAutuSplice.sequence.status.nextStep := #JOB_20_STEP_22;
   END_IF;
END_REGION

REGION Network 89: Step[2022] : Uw Semi Splicer Vacuum Bottm & Uw Semi Splicer Vacuum Top HomePos Command
   RUNG wire#powerrail
      { S7_Templates := "SrcType := DInt" } EQ_Contact(in1 := "Unit1.Em2.ControlNodes".SemiAutuSplice.sequence.status.currentStep, in2 := #JOB_20_STEP_22)
      Contact( "Unit1.Em2.ControlNodes".SemiAutuSplice.sequence.status.seqActive )
      wire#w1
      Contact( "Unit1.EmNodes".emFeedback[0].isLinked )
      I_Contact( "Unit1.EmNodes".emFeedback[1].isLinked )
      wire#w2
      I_Contact( "Unit1.Em2.ControlNodes".cmUwSemiSplicerVacuumRightTopOnOff.monitoring.inHomePos )
      wire#w3
      Coil( "Unit1.Em2.ControlNodes".SemiAutuSplice."step".action[2022] )
   END_RUNG
   RUNG wire#w2
      I_Contact( "Unit1.Em2.ControlNodes".cmUwSemiSplicerVacuumLeftBottomOnOff.monitoring.inHomePos )
   END_RUNG wire#w3
   RUNG wire#w2
      Contact( "Unit1.Em2.ControlNodes".cmUwSemiSplicerVacuumRightTopOnOff.monitoring.inHomePos )
      Contact( "Unit1.Em2.ControlNodes".cmUwSemiSplicerVacuumLeftBottomOnOff.monitoring.inHomePos )
      Coil( "Unit1.Em2.ControlNodes".SemiAutuSplice."step".transition[2022] )
   END_RUNG
   RUNG wire#w2
      Contact( "Unit1.Em2.ControlNodes".SemiAutuSplice."step".transition[2022] )
      { S7_Templates := "time_type := Time" } #statTonTimer[2022].TON(pt := #SeqDelayTime, et =>)
      Move(in := #JOB_20_STEP_25, out1 => "Unit1.Em2.ControlNodes".SemiAutuSplice.sequence.status.nextStep)
   END_RUNG
   RUNG wire#w1
      Contact( "Unit1.EmNodes".emFeedback[1].isLinked )
      I_Contact( "Unit1.EmNodes".emFeedback[0].isLinked )
      wire#w4
      I_Contact( "Unit1.Em2.ControlNodes".cmUwSemiSplicerVacuumRightBottomOnOff.monitoring.inHomePos )
      wire#w5
      Coil( "Unit1.Em2.ControlNodes".SemiAutuSplice."step".action[2023] )
   END_RUNG
   RUNG wire#w4
      I_Contact( "Unit1.Em2.ControlNodes".cmUwSemiSplicerVacuumLeftTopOnOff.monitoring.inHomePos )
   END_RUNG wire#w5
   RUNG wire#w4
      Contact( "Unit1.Em2.ControlNodes".cmUwSemiSplicerVacuumRightBottomOnOff.monitoring.inHomePos )
      Contact( "Unit1.Em2.ControlNodes".cmUwSemiSplicerVacuumLeftTopOnOff.monitoring.inHomePos )
      Coil( "Unit1.Em2.ControlNodes".SemiAutuSplice."step".transition[2023] )
   END_RUNG
   RUNG wire#w4
      Contact( "Unit1.Em2.ControlNodes".SemiAutuSplice."step".transition[2023] )
      { S7_Templates := "time_type := Time" } #statTonTimer[2023].TON(pt := #SeqDelayTime, et =>)
      Move(in := #JOB_20_STEP_25, out1 => "Unit1.Em2.ControlNodes".SemiAutuSplice.sequence.status.nextStep)
   END_RUNG
   // the same network as SCL:
   #_w1 := ("Unit1.Em2.ControlNodes".SemiAutuSplice.sequence.status.currentStep = #JOB_20_STEP_22) AND "Unit1.Em2.ControlNodes".SemiAutuSplice.sequence.status.seqActive;
   #_w2 := #_w1 AND "Unit1.EmNodes".emFeedback[0].isLinked AND NOT "Unit1.EmNodes".emFeedback[1].isLinked;
   "Unit1.Em2.ControlNodes".SemiAutuSplice."step".action[2022] := #_w2 AND (NOT "Unit1.Em2.ControlNodes".cmUwSemiSplicerVacuumRightTopOnOff.monitoring.inHomePos OR NOT "Unit1.Em2.ControlNodes".cmUwSemiSplicerVacuumLeftBottomOnOff.monitoring.inHomePos);
   "Unit1.Em2.ControlNodes".SemiAutuSplice."step".transition[2022] := #_w2 AND "Unit1.Em2.ControlNodes".cmUwSemiSplicerVacuumRightTopOnOff.monitoring.inHomePos AND "Unit1.Em2.ControlNodes".cmUwSemiSplicerVacuumLeftBottomOnOff.monitoring.inHomePos;
   #statTonTimer[2022].TON(IN := #_w2 AND "Unit1.Em2.ControlNodes".SemiAutuSplice."step".transition[2022],
                           PT := #SeqDelayTime);
   IF #statTonTimer[2022].Q THEN
       "Unit1.Em2.ControlNodes".SemiAutuSplice.sequence.status.nextStep := #JOB_20_STEP_25;
   END_IF;
   #_w3 := #_w1 AND "Unit1.EmNodes".emFeedback[1].isLinked AND NOT "Unit1.EmNodes".emFeedback[0].isLinked;
   "Unit1.Em2.ControlNodes".SemiAutuSplice."step".action[2023] := #_w3 AND (NOT "Unit1.Em2.ControlNodes".cmUwSemiSplicerVacuumRightBottomOnOff.monitoring.inHomePos OR NOT "Unit1.Em2.ControlNodes".cmUwSemiSplicerVacuumLeftTopOnOff.monitoring.inHomePos);
   "Unit1.Em2.ControlNodes".SemiAutuSplice."step".transition[2023] := #_w3 AND "Unit1.Em2.ControlNodes".cmUwSemiSplicerVacuumRightBottomOnOff.monitoring.inHomePos AND "Unit1.Em2.ControlNodes".cmUwSemiSplicerVacuumLeftTopOnOff.monitoring.inHomePos;
   #statTonTimer[2023].TON(IN := #_w3 AND "Unit1.Em2.ControlNodes".SemiAutuSplice."step".transition[2023],
                           PT := #SeqDelayTime);
   IF #statTonTimer[2023].Q THEN
       "Unit1.Em2.ControlNodes".SemiAutuSplice.sequence.status.nextStep := #JOB_20_STEP_25;
   END_IF;
END_REGION

REGION Network 90: Step[2025] : Unwinder Axis-B Rewinding & Electrode Holder Mover HomePos Command
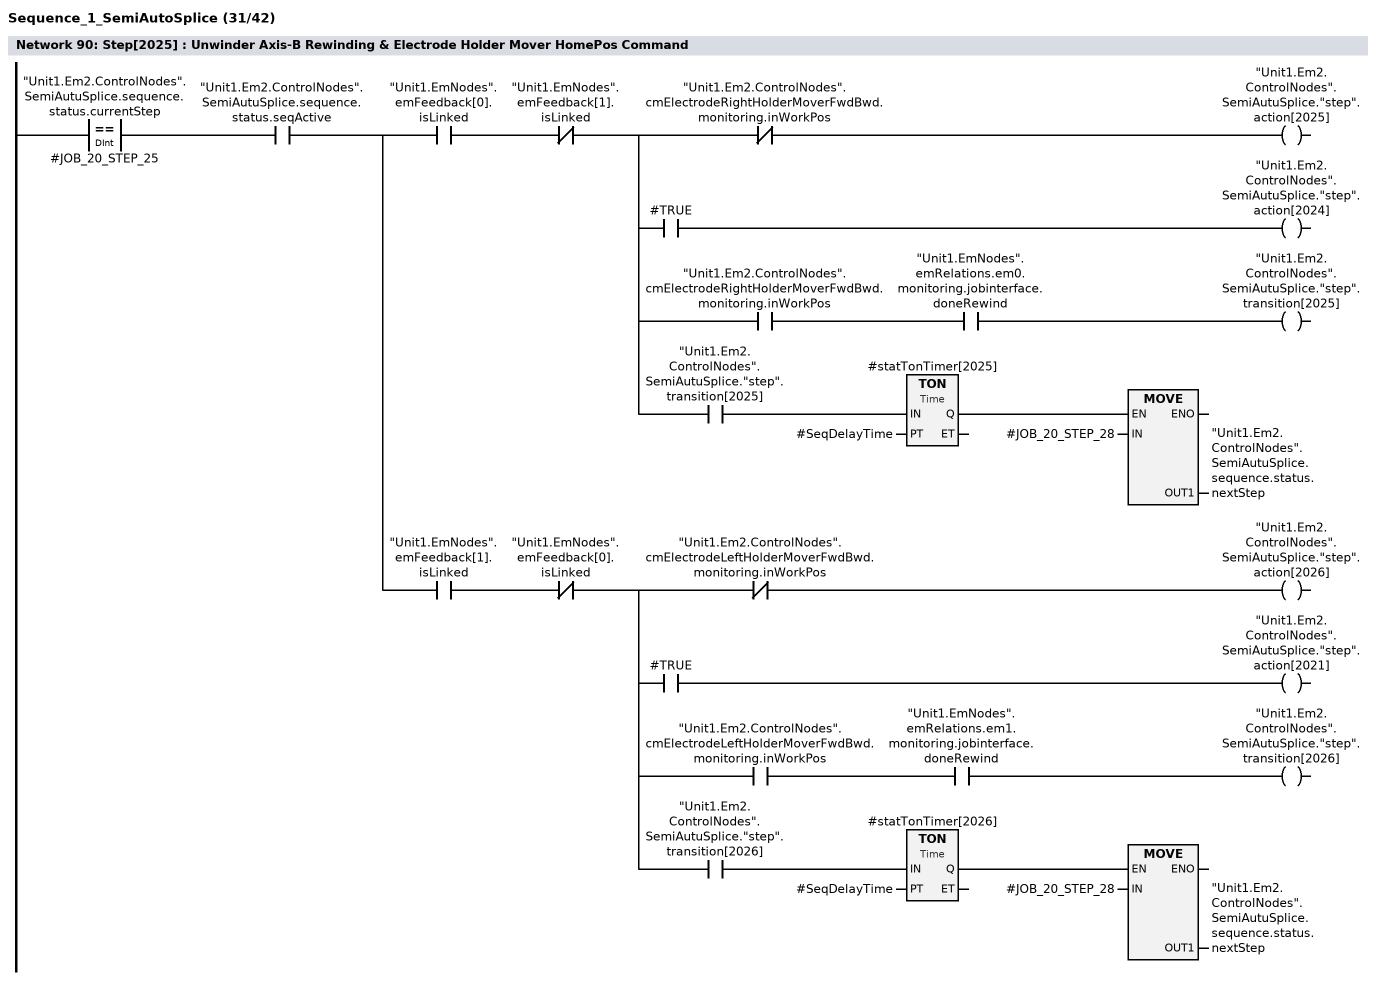
   RUNG wire#powerrail
      { S7_Templates := "SrcType := DInt" } EQ_Contact(in1 := "Unit1.Em2.ControlNodes".SemiAutuSplice.sequence.status.currentStep, in2 := #JOB_20_STEP_25)
      Contact( "Unit1.Em2.ControlNodes".SemiAutuSplice.sequence.status.seqActive )
      wire#w1
      Contact( "Unit1.EmNodes".emFeedback[0].isLinked )
      I_Contact( "Unit1.EmNodes".emFeedback[1].isLinked )
      wire#w2
      I_Contact( "Unit1.Em2.ControlNodes".cmElectrodeRightHolderMoverFwdBwd.monitoring.inWorkPos )
      Coil( "Unit1.Em2.ControlNodes".SemiAutuSplice."step".action[2025] )
   END_RUNG
   RUNG wire#w2
      Contact( #TRUE )
      Coil( "Unit1.Em2.ControlNodes".SemiAutuSplice."step".action[2024] )
   END_RUNG
   RUNG wire#w2
      Contact( "Unit1.Em2.ControlNodes".cmElectrodeRightHolderMoverFwdBwd.monitoring.inWorkPos )
      Contact( "Unit1.EmNodes".emRelations.em0.monitoring.jobinterface.doneRewind )
      Coil( "Unit1.Em2.ControlNodes".SemiAutuSplice."step".transition[2025] )
   END_RUNG
   RUNG wire#w2
      Contact( "Unit1.Em2.ControlNodes".SemiAutuSplice."step".transition[2025] )
      { S7_Templates := "time_type := Time" } #statTonTimer[2025].TON(pt := #SeqDelayTime, et =>)
      Move(in := #JOB_20_STEP_28, out1 => "Unit1.Em2.ControlNodes".SemiAutuSplice.sequence.status.nextStep)
   END_RUNG
   RUNG wire#w1
      Contact( "Unit1.EmNodes".emFeedback[1].isLinked )
      I_Contact( "Unit1.EmNodes".emFeedback[0].isLinked )
      wire#w3
      I_Contact( "Unit1.Em2.ControlNodes".cmElectrodeLeftHolderMoverFwdBwd.monitoring.inWorkPos )
      Coil( "Unit1.Em2.ControlNodes".SemiAutuSplice."step".action[2026] )
   END_RUNG
   RUNG wire#w3
      Contact( #TRUE )
      Coil( "Unit1.Em2.ControlNodes".SemiAutuSplice."step".action[2021] )
   END_RUNG
   RUNG wire#w3
      Contact( "Unit1.Em2.ControlNodes".cmElectrodeLeftHolderMoverFwdBwd.monitoring.inWorkPos )
      Contact( "Unit1.EmNodes".emRelations.em1.monitoring.jobinterface.doneRewind )
      Coil( "Unit1.Em2.ControlNodes".SemiAutuSplice."step".transition[2026] )
   END_RUNG
   RUNG wire#w3
      Contact( "Unit1.Em2.ControlNodes".SemiAutuSplice."step".transition[2026] )
      { S7_Templates := "time_type := Time" } #statTonTimer[2026].TON(pt := #SeqDelayTime, et =>)
      Move(in := #JOB_20_STEP_28, out1 => "Unit1.Em2.ControlNodes".SemiAutuSplice.sequence.status.nextStep)
   END_RUNG
   // the same network as SCL:
   #_w1 := ("Unit1.Em2.ControlNodes".SemiAutuSplice.sequence.status.currentStep = #JOB_20_STEP_25) AND "Unit1.Em2.ControlNodes".SemiAutuSplice.sequence.status.seqActive;
   #_w2 := #_w1 AND "Unit1.EmNodes".emFeedback[0].isLinked AND NOT "Unit1.EmNodes".emFeedback[1].isLinked;
   "Unit1.Em2.ControlNodes".SemiAutuSplice."step".action[2025] := #_w2 AND NOT "Unit1.Em2.ControlNodes".cmElectrodeRightHolderMoverFwdBwd.monitoring.inWorkPos;
   "Unit1.Em2.ControlNodes".SemiAutuSplice."step".action[2024] := #_w2 AND #TRUE;
   "Unit1.Em2.ControlNodes".SemiAutuSplice."step".transition[2025] := #_w2 AND "Unit1.Em2.ControlNodes".cmElectrodeRightHolderMoverFwdBwd.monitoring.inWorkPos AND "Unit1.EmNodes".emRelations.em0.monitoring.jobinterface.doneRewind;
   #statTonTimer[2025].TON(IN := #_w2 AND "Unit1.Em2.ControlNodes".SemiAutuSplice."step".transition[2025],
                           PT := #SeqDelayTime);
   IF #statTonTimer[2025].Q THEN
       "Unit1.Em2.ControlNodes".SemiAutuSplice.sequence.status.nextStep := #JOB_20_STEP_28;
   END_IF;
   #_w3 := #_w1 AND "Unit1.EmNodes".emFeedback[1].isLinked AND NOT "Unit1.EmNodes".emFeedback[0].isLinked;
   "Unit1.Em2.ControlNodes".SemiAutuSplice."step".action[2026] := #_w3 AND NOT "Unit1.Em2.ControlNodes".cmElectrodeLeftHolderMoverFwdBwd.monitoring.inWorkPos;
   "Unit1.Em2.ControlNodes".SemiAutuSplice."step".action[2021] := #_w3 AND #TRUE;
   "Unit1.Em2.ControlNodes".SemiAutuSplice."step".transition[2026] := #_w3 AND "Unit1.Em2.ControlNodes".cmElectrodeLeftHolderMoverFwdBwd.monitoring.inWorkPos AND "Unit1.EmNodes".emRelations.em1.monitoring.jobinterface.doneRewind;
   #statTonTimer[2026].TON(IN := #_w3 AND "Unit1.Em2.ControlNodes".SemiAutuSplice."step".transition[2026],
                           PT := #SeqDelayTime);
   IF #statTonTimer[2026].Q THEN
       "Unit1.Em2.ControlNodes".SemiAutuSplice.sequence.status.nextStep := #JOB_20_STEP_28;
   END_IF;
END_REGION

REGION Network 91: Step[2028] : Uw Semi Splicer Vaccum Top HomePos & Uw Semi Splicer Top WorkPos Command
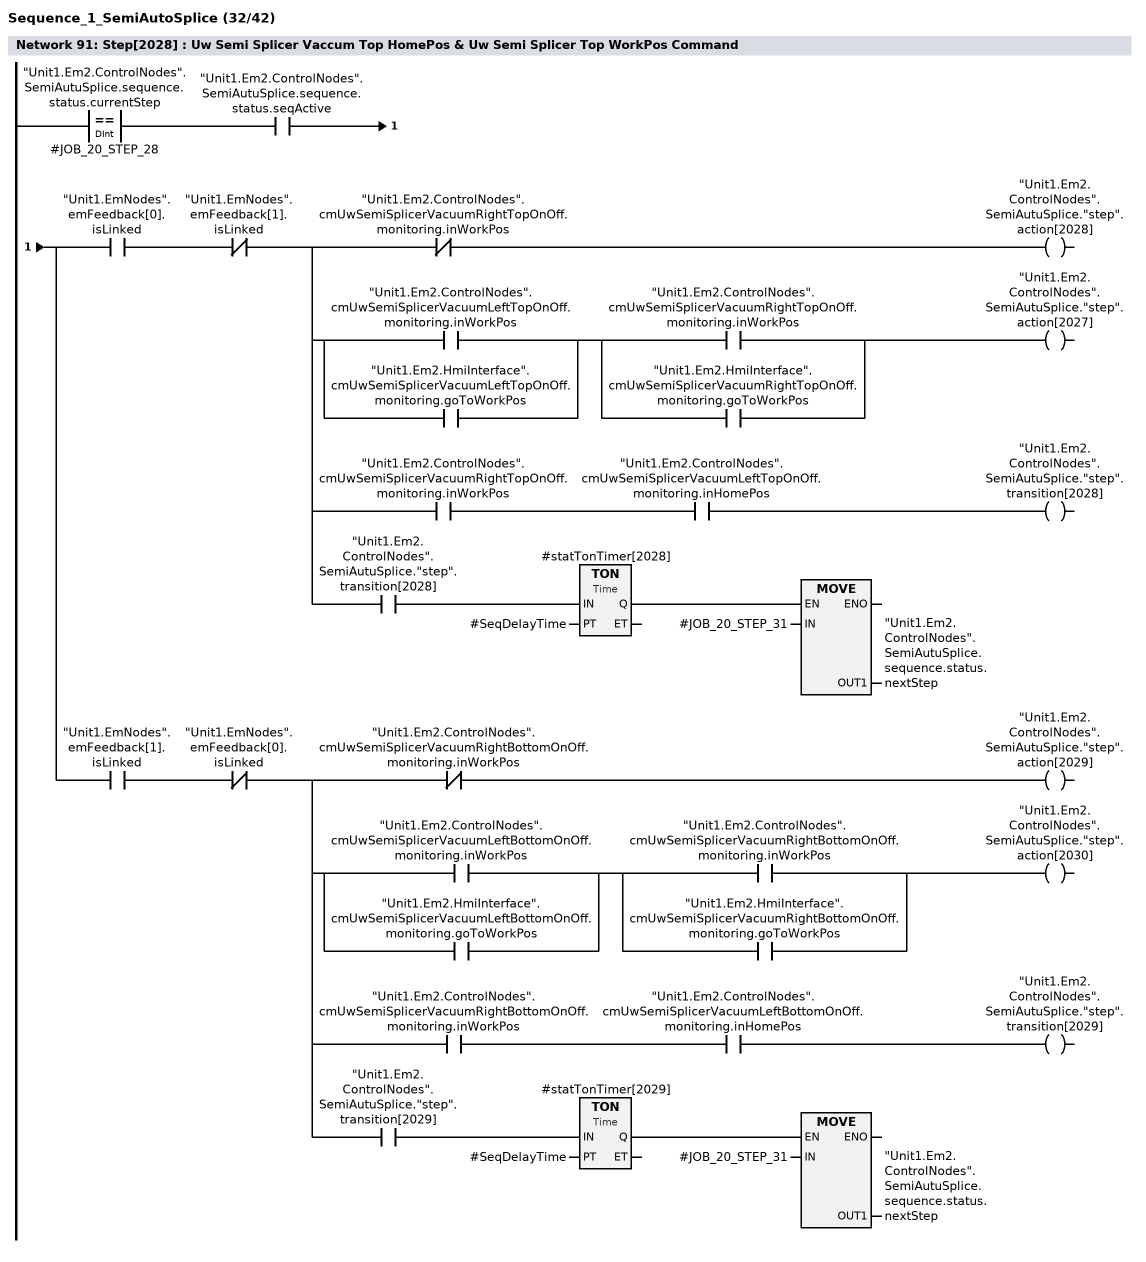
   RUNG wire#powerrail
      { S7_Templates := "SrcType := DInt" } EQ_Contact(in1 := "Unit1.Em2.ControlNodes".SemiAutuSplice.sequence.status.currentStep, in2 := #JOB_20_STEP_28)
      Contact( "Unit1.Em2.ControlNodes".SemiAutuSplice.sequence.status.seqActive )
      wire#w1
      Contact( "Unit1.EmNodes".emFeedback[0].isLinked )
      I_Contact( "Unit1.EmNodes".emFeedback[1].isLinked )
      wire#w2
      I_Contact( "Unit1.Em2.ControlNodes".cmUwSemiSplicerVacuumRightTopOnOff.monitoring.inWorkPos )
      Coil( "Unit1.Em2.ControlNodes".SemiAutuSplice."step".action[2028] )
   END_RUNG
   RUNG wire#w2
      Contact( "Unit1.Em2.ControlNodes".cmUwSemiSplicerVacuumLeftTopOnOff.monitoring.inWorkPos )
      wire#w3
      Contact( "Unit1.Em2.ControlNodes".cmUwSemiSplicerVacuumRightTopOnOff.monitoring.inWorkPos )
      wire#w4
      Coil( "Unit1.Em2.ControlNodes".SemiAutuSplice."step".action[2027] )
   END_RUNG
   RUNG wire#w2
      Contact( "Unit1.Em2.HmiInterface".cmUwSemiSplicerVacuumLeftTopOnOff.monitoring.goToWorkPos )
   END_RUNG wire#w3
   RUNG wire#w3
      Contact( "Unit1.Em2.HmiInterface".cmUwSemiSplicerVacuumRightTopOnOff.monitoring.goToWorkPos )
   END_RUNG wire#w4
   RUNG wire#w2
      Contact( "Unit1.Em2.ControlNodes".cmUwSemiSplicerVacuumRightTopOnOff.monitoring.inWorkPos )
      Contact( "Unit1.Em2.ControlNodes".cmUwSemiSplicerVacuumLeftTopOnOff.monitoring.inHomePos )
      Coil( "Unit1.Em2.ControlNodes".SemiAutuSplice."step".transition[2028] )
   END_RUNG
   RUNG wire#w2
      Contact( "Unit1.Em2.ControlNodes".SemiAutuSplice."step".transition[2028] )
      { S7_Templates := "time_type := Time" } #statTonTimer[2028].TON(pt := #SeqDelayTime, et =>)
      Move(in := #JOB_20_STEP_31, out1 => "Unit1.Em2.ControlNodes".SemiAutuSplice.sequence.status.nextStep)
   END_RUNG
   RUNG wire#w1
      Contact( "Unit1.EmNodes".emFeedback[1].isLinked )
      I_Contact( "Unit1.EmNodes".emFeedback[0].isLinked )
      wire#w5
      I_Contact( "Unit1.Em2.ControlNodes".cmUwSemiSplicerVacuumRightBottomOnOff.monitoring.inWorkPos )
      Coil( "Unit1.Em2.ControlNodes".SemiAutuSplice."step".action[2029] )
   END_RUNG
   RUNG wire#w5
      Contact( "Unit1.Em2.ControlNodes".cmUwSemiSplicerVacuumLeftBottomOnOff.monitoring.inWorkPos )
      wire#w6
      Contact( "Unit1.Em2.ControlNodes".cmUwSemiSplicerVacuumRightBottomOnOff.monitoring.inWorkPos )
      wire#w7
      Coil( "Unit1.Em2.ControlNodes".SemiAutuSplice."step".action[2030] )
   END_RUNG
   RUNG wire#w5
      Contact( "Unit1.Em2.HmiInterface".cmUwSemiSplicerVacuumLeftBottomOnOff.monitoring.goToWorkPos )
   END_RUNG wire#w6
   RUNG wire#w6
      Contact( "Unit1.Em2.HmiInterface".cmUwSemiSplicerVacuumRightBottomOnOff.monitoring.goToWorkPos )
   END_RUNG wire#w7
   RUNG wire#w5
      Contact( "Unit1.Em2.ControlNodes".cmUwSemiSplicerVacuumRightBottomOnOff.monitoring.inWorkPos )
      Contact( "Unit1.Em2.ControlNodes".cmUwSemiSplicerVacuumLeftBottomOnOff.monitoring.inHomePos )
      Coil( "Unit1.Em2.ControlNodes".SemiAutuSplice."step".transition[2029] )
   END_RUNG
   RUNG wire#w5
      Contact( "Unit1.Em2.ControlNodes".SemiAutuSplice."step".transition[2029] )
      { S7_Templates := "time_type := Time" } #statTonTimer[2029].TON(pt := #SeqDelayTime, et =>)
      Move(in := #JOB_20_STEP_31, out1 => "Unit1.Em2.ControlNodes".SemiAutuSplice.sequence.status.nextStep)
   END_RUNG
   // the same network as SCL:
   #_w1 := ("Unit1.Em2.ControlNodes".SemiAutuSplice.sequence.status.currentStep = #JOB_20_STEP_28) AND "Unit1.Em2.ControlNodes".SemiAutuSplice.sequence.status.seqActive;
   #_w2 := #_w1 AND "Unit1.EmNodes".emFeedback[0].isLinked AND NOT "Unit1.EmNodes".emFeedback[1].isLinked;
   "Unit1.Em2.ControlNodes".SemiAutuSplice."step".action[2028] := #_w2 AND NOT "Unit1.Em2.ControlNodes".cmUwSemiSplicerVacuumRightTopOnOff.monitoring.inWorkPos;
   "Unit1.Em2.ControlNodes".SemiAutuSplice."step".action[2027] := #_w2 AND ("Unit1.Em2.ControlNodes".cmUwSemiSplicerVacuumLeftTopOnOff.monitoring.inWorkPos OR "Unit1.Em2.HmiInterface".cmUwSemiSplicerVacuumLeftTopOnOff.monitoring.goToWorkPos) AND ("Unit1.Em2.ControlNodes".cmUwSemiSplicerVacuumRightTopOnOff.monitoring.inWorkPos OR "Unit1.Em2.HmiInterface".cmUwSemiSplicerVacuumRightTopOnOff.monitoring.goToWorkPos);
   "Unit1.Em2.ControlNodes".SemiAutuSplice."step".transition[2028] := #_w2 AND "Unit1.Em2.ControlNodes".cmUwSemiSplicerVacuumRightTopOnOff.monitoring.inWorkPos AND "Unit1.Em2.ControlNodes".cmUwSemiSplicerVacuumLeftTopOnOff.monitoring.inHomePos;
   #statTonTimer[2028].TON(IN := #_w2 AND "Unit1.Em2.ControlNodes".SemiAutuSplice."step".transition[2028],
                           PT := #SeqDelayTime);
   IF #statTonTimer[2028].Q THEN
       "Unit1.Em2.ControlNodes".SemiAutuSplice.sequence.status.nextStep := #JOB_20_STEP_31;
   END_IF;
   #_w3 := #_w1 AND "Unit1.EmNodes".emFeedback[1].isLinked AND NOT "Unit1.EmNodes".emFeedback[0].isLinked;
   "Unit1.Em2.ControlNodes".SemiAutuSplice."step".action[2029] := #_w3 AND NOT "Unit1.Em2.ControlNodes".cmUwSemiSplicerVacuumRightBottomOnOff.monitoring.inWorkPos;
   "Unit1.Em2.ControlNodes".SemiAutuSplice."step".action[2030] := #_w3 AND ("Unit1.Em2.ControlNodes".cmUwSemiSplicerVacuumLeftBottomOnOff.monitoring.inWorkPos OR "Unit1.Em2.HmiInterface".cmUwSemiSplicerVacuumLeftBottomOnOff.monitoring.goToWorkPos) AND ("Unit1.Em2.ControlNodes".cmUwSemiSplicerVacuumRightBottomOnOff.monitoring.inWorkPos OR "Unit1.Em2.HmiInterface".cmUwSemiSplicerVacuumRightBottomOnOff.monitoring.goToWorkPos);
   "Unit1.Em2.ControlNodes".SemiAutuSplice."step".transition[2029] := #_w3 AND "Unit1.Em2.ControlNodes".cmUwSemiSplicerVacuumRightBottomOnOff.monitoring.inWorkPos AND "Unit1.Em2.ControlNodes".cmUwSemiSplicerVacuumLeftBottomOnOff.monitoring.inHomePos;
   #statTonTimer[2029].TON(IN := #_w3 AND "Unit1.Em2.ControlNodes".SemiAutuSplice."step".transition[2029],
                           PT := #SeqDelayTime);
   IF #statTonTimer[2029].Q THEN
       "Unit1.Em2.ControlNodes".SemiAutuSplice.sequence.status.nextStep := #JOB_20_STEP_31;
   END_IF;
END_REGION

REGION Network 92: Step[2031] : Electrode Fix Top & Electrode Fix Bottom HomePos Command
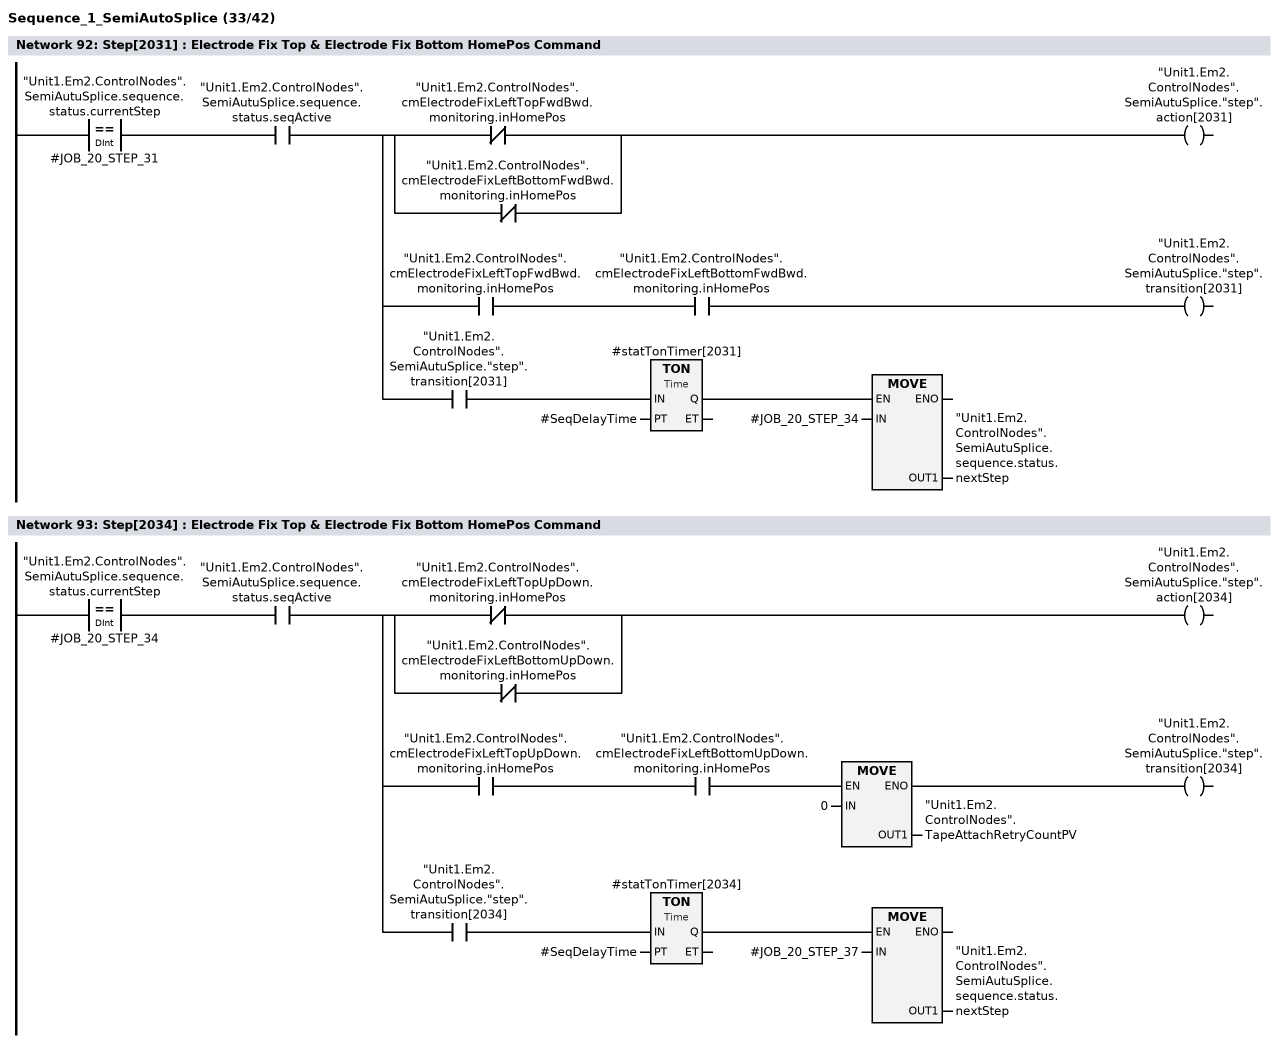
   RUNG wire#powerrail
      { S7_Templates := "SrcType := DInt" } EQ_Contact(in1 := "Unit1.Em2.ControlNodes".SemiAutuSplice.sequence.status.currentStep, in2 := #JOB_20_STEP_31)
      Contact( "Unit1.Em2.ControlNodes".SemiAutuSplice.sequence.status.seqActive )
      wire#w1
      I_Contact( "Unit1.Em2.ControlNodes".cmElectrodeFixLeftTopFwdBwd.monitoring.inHomePos )
      wire#w2
      Coil( "Unit1.Em2.ControlNodes".SemiAutuSplice."step".action[2031] )
   END_RUNG
   RUNG wire#w1
      I_Contact( "Unit1.Em2.ControlNodes".cmElectrodeFixLeftBottomFwdBwd.monitoring.inHomePos )
   END_RUNG wire#w2
   RUNG wire#w1
      Contact( "Unit1.Em2.ControlNodes".cmElectrodeFixLeftTopFwdBwd.monitoring.inHomePos )
      Contact( "Unit1.Em2.ControlNodes".cmElectrodeFixLeftBottomFwdBwd.monitoring.inHomePos )
      Coil( "Unit1.Em2.ControlNodes".SemiAutuSplice."step".transition[2031] )
   END_RUNG
   RUNG wire#w1
      Contact( "Unit1.Em2.ControlNodes".SemiAutuSplice."step".transition[2031] )
      { S7_Templates := "time_type := Time" } #statTonTimer[2031].TON(pt := #SeqDelayTime, et =>)
      Move(in := #JOB_20_STEP_34, out1 => "Unit1.Em2.ControlNodes".SemiAutuSplice.sequence.status.nextStep)
   END_RUNG
   // the same network as SCL:
   #_w1 := ("Unit1.Em2.ControlNodes".SemiAutuSplice.sequence.status.currentStep = #JOB_20_STEP_31) AND "Unit1.Em2.ControlNodes".SemiAutuSplice.sequence.status.seqActive;
   "Unit1.Em2.ControlNodes".SemiAutuSplice."step".action[2031] := #_w1 AND (NOT "Unit1.Em2.ControlNodes".cmElectrodeFixLeftTopFwdBwd.monitoring.inHomePos OR NOT "Unit1.Em2.ControlNodes".cmElectrodeFixLeftBottomFwdBwd.monitoring.inHomePos);
   "Unit1.Em2.ControlNodes".SemiAutuSplice."step".transition[2031] := #_w1 AND "Unit1.Em2.ControlNodes".cmElectrodeFixLeftTopFwdBwd.monitoring.inHomePos AND "Unit1.Em2.ControlNodes".cmElectrodeFixLeftBottomFwdBwd.monitoring.inHomePos;
   #statTonTimer[2031].TON(IN := #_w1 AND "Unit1.Em2.ControlNodes".SemiAutuSplice."step".transition[2031],
                           PT := #SeqDelayTime);
   IF #statTonTimer[2031].Q THEN
       "Unit1.Em2.ControlNodes".SemiAutuSplice.sequence.status.nextStep := #JOB_20_STEP_34;
   END_IF;
END_REGION

REGION Network 93: Step[2034] : Electrode Fix Top & Electrode Fix Bottom HomePos Command
   RUNG wire#powerrail
      { S7_Templates := "SrcType := DInt" } EQ_Contact(in1 := "Unit1.Em2.ControlNodes".SemiAutuSplice.sequence.status.currentStep, in2 := #JOB_20_STEP_34)
      Contact( "Unit1.Em2.ControlNodes".SemiAutuSplice.sequence.status.seqActive )
      wire#w1
      I_Contact( "Unit1.Em2.ControlNodes".cmElectrodeFixLeftTopUpDown.monitoring.inHomePos )
      wire#w2
      Coil( "Unit1.Em2.ControlNodes".SemiAutuSplice."step".action[2034] )
   END_RUNG
   RUNG wire#w1
      I_Contact( "Unit1.Em2.ControlNodes".cmElectrodeFixLeftBottomUpDown.monitoring.inHomePos )
   END_RUNG wire#w2
   RUNG wire#w1
      Contact( "Unit1.Em2.ControlNodes".cmElectrodeFixLeftTopUpDown.monitoring.inHomePos )
      Contact( "Unit1.Em2.ControlNodes".cmElectrodeFixLeftBottomUpDown.monitoring.inHomePos )
      Move(in := 0, out1 => "Unit1.Em2.ControlNodes".TapeAttachRetryCountPV)
      Coil( "Unit1.Em2.ControlNodes".SemiAutuSplice."step".transition[2034] )
   END_RUNG
   RUNG wire#w1
      Contact( "Unit1.Em2.ControlNodes".SemiAutuSplice."step".transition[2034] )
      { S7_Templates := "time_type := Time" } #statTonTimer[2034].TON(pt := #SeqDelayTime, et =>)
      Move(in := #JOB_20_STEP_37, out1 => "Unit1.Em2.ControlNodes".SemiAutuSplice.sequence.status.nextStep)
   END_RUNG
   // the same network as SCL:
   #_w1 := ("Unit1.Em2.ControlNodes".SemiAutuSplice.sequence.status.currentStep = #JOB_20_STEP_34) AND "Unit1.Em2.ControlNodes".SemiAutuSplice.sequence.status.seqActive;
   "Unit1.Em2.ControlNodes".SemiAutuSplice."step".action[2034] := #_w1 AND (NOT "Unit1.Em2.ControlNodes".cmElectrodeFixLeftTopUpDown.monitoring.inHomePos OR NOT "Unit1.Em2.ControlNodes".cmElectrodeFixLeftBottomUpDown.monitoring.inHomePos);
   #_w2 := #_w1 AND "Unit1.Em2.ControlNodes".cmElectrodeFixLeftTopUpDown.monitoring.inHomePos AND "Unit1.Em2.ControlNodes".cmElectrodeFixLeftBottomUpDown.monitoring.inHomePos;
   IF #_w2 THEN "Unit1.Em2.ControlNodes".TapeAttachRetryCountPV := 0; END_IF;
   "Unit1.Em2.ControlNodes".SemiAutuSplice."step".transition[2034] := #_w2;
   #statTonTimer[2034].TON(IN := #_w1 AND "Unit1.Em2.ControlNodes".SemiAutuSplice."step".transition[2034],
                           PT := #SeqDelayTime);
   IF #statTonTimer[2034].Q THEN
       "Unit1.Em2.ControlNodes".SemiAutuSplice.sequence.status.nextStep := #JOB_20_STEP_37;
   END_IF;
END_REGION

REGION Network 94: Step[2037] : Tape Loading Turn WorkPos Command
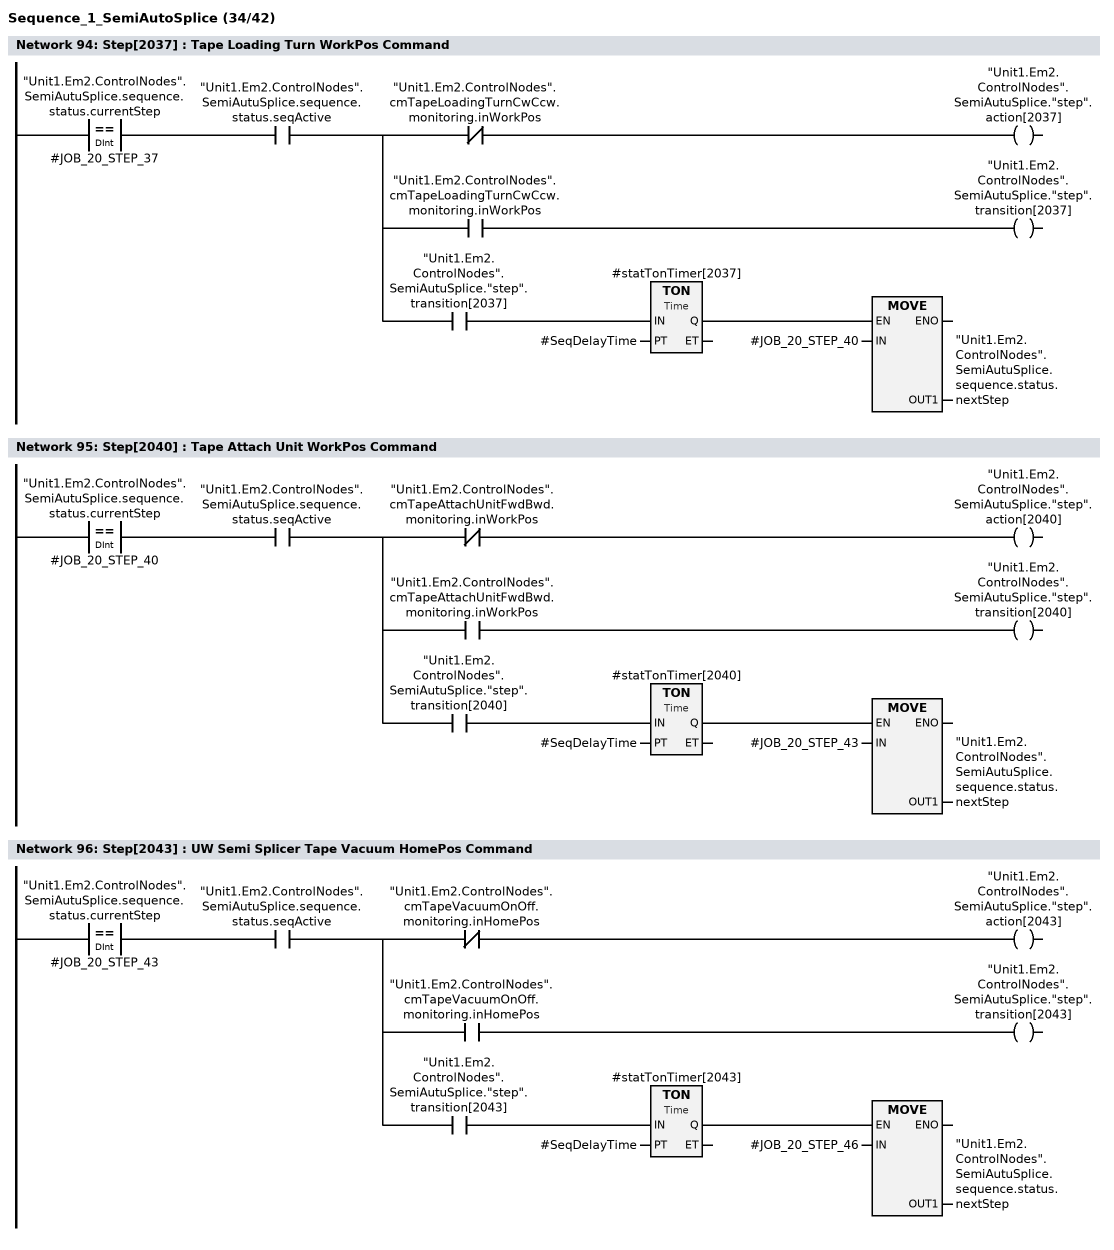
   RUNG wire#powerrail
      { S7_Templates := "SrcType := DInt" } EQ_Contact(in1 := "Unit1.Em2.ControlNodes".SemiAutuSplice.sequence.status.currentStep, in2 := #JOB_20_STEP_37)
      Contact( "Unit1.Em2.ControlNodes".SemiAutuSplice.sequence.status.seqActive )
      wire#w1
      I_Contact( "Unit1.Em2.ControlNodes".cmTapeLoadingTurnCwCcw.monitoring.inWorkPos )
      Coil( "Unit1.Em2.ControlNodes".SemiAutuSplice."step".action[2037] )
   END_RUNG
   RUNG wire#w1
      Contact( "Unit1.Em2.ControlNodes".cmTapeLoadingTurnCwCcw.monitoring.inWorkPos )
      Coil( "Unit1.Em2.ControlNodes".SemiAutuSplice."step".transition[2037] )
   END_RUNG
   RUNG wire#w1
      Contact( "Unit1.Em2.ControlNodes".SemiAutuSplice."step".transition[2037] )
      { S7_Templates := "time_type := Time" } #statTonTimer[2037].TON(pt := #SeqDelayTime, et =>)
      Move(in := #JOB_20_STEP_40, out1 => "Unit1.Em2.ControlNodes".SemiAutuSplice.sequence.status.nextStep)
   END_RUNG
   // the same network as SCL:
   #_w1 := ("Unit1.Em2.ControlNodes".SemiAutuSplice.sequence.status.currentStep = #JOB_20_STEP_37) AND "Unit1.Em2.ControlNodes".SemiAutuSplice.sequence.status.seqActive;
   "Unit1.Em2.ControlNodes".SemiAutuSplice."step".action[2037] := #_w1 AND NOT "Unit1.Em2.ControlNodes".cmTapeLoadingTurnCwCcw.monitoring.inWorkPos;
   "Unit1.Em2.ControlNodes".SemiAutuSplice."step".transition[2037] := #_w1 AND "Unit1.Em2.ControlNodes".cmTapeLoadingTurnCwCcw.monitoring.inWorkPos;
   #statTonTimer[2037].TON(IN := #_w1 AND "Unit1.Em2.ControlNodes".SemiAutuSplice."step".transition[2037],
                           PT := #SeqDelayTime);
   IF #statTonTimer[2037].Q THEN
       "Unit1.Em2.ControlNodes".SemiAutuSplice.sequence.status.nextStep := #JOB_20_STEP_40;
   END_IF;
END_REGION

REGION Network 95: Step[2040] : Tape Attach Unit WorkPos Command
   RUNG wire#powerrail
      { S7_Templates := "SrcType := DInt" } EQ_Contact(in1 := "Unit1.Em2.ControlNodes".SemiAutuSplice.sequence.status.currentStep, in2 := #JOB_20_STEP_40)
      Contact( "Unit1.Em2.ControlNodes".SemiAutuSplice.sequence.status.seqActive )
      wire#w1
      I_Contact( "Unit1.Em2.ControlNodes".cmTapeAttachUnitFwdBwd.monitoring.inWorkPos )
      Coil( "Unit1.Em2.ControlNodes".SemiAutuSplice."step".action[2040] )
   END_RUNG
   RUNG wire#w1
      Contact( "Unit1.Em2.ControlNodes".cmTapeAttachUnitFwdBwd.monitoring.inWorkPos )
      Coil( "Unit1.Em2.ControlNodes".SemiAutuSplice."step".transition[2040] )
   END_RUNG
   RUNG wire#w1
      Contact( "Unit1.Em2.ControlNodes".SemiAutuSplice."step".transition[2040] )
      { S7_Templates := "time_type := Time" } #statTonTimer[2040].TON(pt := #SeqDelayTime, et =>)
      Move(in := #JOB_20_STEP_43, out1 => "Unit1.Em2.ControlNodes".SemiAutuSplice.sequence.status.nextStep)
   END_RUNG
   // the same network as SCL:
   #_w1 := ("Unit1.Em2.ControlNodes".SemiAutuSplice.sequence.status.currentStep = #JOB_20_STEP_40) AND "Unit1.Em2.ControlNodes".SemiAutuSplice.sequence.status.seqActive;
   "Unit1.Em2.ControlNodes".SemiAutuSplice."step".action[2040] := #_w1 AND NOT "Unit1.Em2.ControlNodes".cmTapeAttachUnitFwdBwd.monitoring.inWorkPos;
   "Unit1.Em2.ControlNodes".SemiAutuSplice."step".transition[2040] := #_w1 AND "Unit1.Em2.ControlNodes".cmTapeAttachUnitFwdBwd.monitoring.inWorkPos;
   #statTonTimer[2040].TON(IN := #_w1 AND "Unit1.Em2.ControlNodes".SemiAutuSplice."step".transition[2040],
                           PT := #SeqDelayTime);
   IF #statTonTimer[2040].Q THEN
       "Unit1.Em2.ControlNodes".SemiAutuSplice.sequence.status.nextStep := #JOB_20_STEP_43;
   END_IF;
END_REGION

REGION Network 96: Step[2043] : UW Semi Splicer Tape Vacuum HomePos Command
   RUNG wire#powerrail
      { S7_Templates := "SrcType := DInt" } EQ_Contact(in1 := "Unit1.Em2.ControlNodes".SemiAutuSplice.sequence.status.currentStep, in2 := #JOB_20_STEP_43)
      Contact( "Unit1.Em2.ControlNodes".SemiAutuSplice.sequence.status.seqActive )
      wire#w1
      I_Contact( "Unit1.Em2.ControlNodes".cmTapeVacuumOnOff.monitoring.inHomePos )
      Coil( "Unit1.Em2.ControlNodes".SemiAutuSplice."step".action[2043] )
   END_RUNG
   RUNG wire#w1
      Contact( "Unit1.Em2.ControlNodes".cmTapeVacuumOnOff.monitoring.inHomePos )
      Coil( "Unit1.Em2.ControlNodes".SemiAutuSplice."step".transition[2043] )
   END_RUNG
   RUNG wire#w1
      Contact( "Unit1.Em2.ControlNodes".SemiAutuSplice."step".transition[2043] )
      { S7_Templates := "time_type := Time" } #statTonTimer[2043].TON(pt := #SeqDelayTime, et =>)
      Move(in := #JOB_20_STEP_46, out1 => "Unit1.Em2.ControlNodes".SemiAutuSplice.sequence.status.nextStep)
   END_RUNG
   // the same network as SCL:
   #_w1 := ("Unit1.Em2.ControlNodes".SemiAutuSplice.sequence.status.currentStep = #JOB_20_STEP_43) AND "Unit1.Em2.ControlNodes".SemiAutuSplice.sequence.status.seqActive;
   "Unit1.Em2.ControlNodes".SemiAutuSplice."step".action[2043] := #_w1 AND NOT "Unit1.Em2.ControlNodes".cmTapeVacuumOnOff.monitoring.inHomePos;
   "Unit1.Em2.ControlNodes".SemiAutuSplice."step".transition[2043] := #_w1 AND "Unit1.Em2.ControlNodes".cmTapeVacuumOnOff.monitoring.inHomePos;
   #statTonTimer[2043].TON(IN := #_w1 AND "Unit1.Em2.ControlNodes".SemiAutuSplice."step".transition[2043],
                           PT := #SeqDelayTime);
   IF #statTonTimer[2043].Q THEN
       "Unit1.Em2.ControlNodes".SemiAutuSplice.sequence.status.nextStep := #JOB_20_STEP_46;
   END_IF;
END_REGION

